DECL FDAT FP437={TOOL_NO 1,BASE_NO 1,IPO_FRAME #BASE,POINT2[] " ",TQ_STATE FALSE}
DECL E6POS XP437={X 1259.09706,Y 164.02997,Z 815.2861,A 180,B 0,C -180,S 2,T 2,E1 0,E2 0,E3 0,E4 0,E5 0,E6 0}
DECL PDAT PPDATP96={VEL 100,ACC 100,APO_DIST 100,APO_MODE #CDIS,GEAR_JERK 100.000,EXAX_IGN 0}
DECL FDAT FP33={TOOL_NO 1,BASE_NO 1,IPO_FRAME #BASE,POINT2[] " ",TQ_STATE FALSE}
DECL E6POS XP33={X 427.07288,Y -471.93323,Z 1236.2934,A 180,B 0,C 180,S 2,T 2,E1 0,E2 0,E3 0,E4 0,E5 0,E6 0}
DECL LDAT LCPDATP186={VEL 1,ACC 100,APO_DIST 100,APO_FAC 50.0,ORI_TYP #VAR,CIRC_TYP #BASE,JERK_FAC 50.0}
DECL FDAT FP31={TOOL_NO 1,BASE_NO 1,IPO_FRAME #BASE,POINT2[] " ",TQ_STATE FALSE}
DECL E6POS XP31={X 427.07317,Y -471.93292,Z 1136.29359,A -180,B 0,C 180,S 2,T 2,E1 0,E2 0,E3 0,E4 0,E5 0,E6 0}
DECL LDAT LCPDATP187={VEL 1,ACC 100,APO_DIST 100,APO_FAC 50.0,ORI_TYP #VAR,CIRC_TYP #BASE,JERK_FAC 50.0}
DECL FDAT FP32={TOOL_NO 1,BASE_NO 1,IPO_FRAME #BASE,POINT2[] " ",TQ_STATE FALSE}
DECL E6POS XP32={X 377.07317,Y -471.93292,Z 1036.29359,A -180,B 0,C 180,S 2,T 2,E1 0,E2 0,E3 0,E4 0,E5 0,E6 0}
; DECL PDAT PPDATP96={VEL 100,ACC 100,APO_DIST 100,APO_MODE #CDIS,GEAR_JERK 100.000,EXAX_IGN 0}
DECL FDAT FP273={TOOL_NO 1,BASE_NO 1,IPO_FRAME #BASE,POINT2[] " ",TQ_STATE FALSE}
DECL E6POS XP273={X 745.07288,Y -471.93323,Z 1236.2934,A 180,B 0,C 180,S 2,T 2,E1 0,E2 0,E3 0,E4 0,E5 0,E6 0}
; DECL LDAT LCPDATP186={VEL 1,ACC 100,APO_DIST 100,APO_FAC 50.0,ORI_TYP #VAR,CIRC_TYP #BASE,JERK_FAC 50.0}
DECL FDAT FP274={TOOL_NO 1,BASE_NO 1,IPO_FRAME #BASE,POINT2[] " ",TQ_STATE FALSE}
DECL E6POS XP274={X 745.07317,Y -471.93292,Z 1136.29359,A -180,B 0,C 180,S 2,T 2,E1 0,E2 0,E3 0,E4 0,E5 0,E6 0}
; DECL LDAT LCPDATP187={VEL 1,ACC 100,APO_DIST 100,APO_FAC 50.0,ORI_TYP #VAR,CIRC_TYP #BASE,JERK_FAC 50.0}
DECL FDAT FP275={TOOL_NO 1,BASE_NO 1,IPO_FRAME #BASE,POINT2[] " ",TQ_STATE FALSE}
DECL E6POS XP275={X 695.07317,Y -471.93292,Z 1036.29359,A -180,B 0,C 180,S 2,T 2,E1 0,E2 0,E3 0,E4 0,E5 0,E6 0}
DECL PDAT PPDATP97={VEL 100,ACC 100,APO_DIST 100,APO_MODE #CDIS,GEAR_JERK 100.000,EXAX_IGN 0}
DECL FDAT FP278={TOOL_NO 1,BASE_NO 1,IPO_FRAME #BASE,POINT2[] " ",TQ_STATE FALSE}
DECL E6POS XP278={X 537.09939,Y -651.74884,Z 1306.29683,A 90,B 0,C 180,S 2,T 2,E1 0,E2 0,E3 0,E4 0,E5 0,E6 0}
DECL LDAT LCPDATP188={VEL 1,ACC 100,APO_DIST 100,APO_FAC 50.0,ORI_TYP #VAR,CIRC_TYP #BASE,JERK_FAC 50.0}
DECL FDAT FP276={TOOL_NO 1,BASE_NO 1,IPO_FRAME #BASE,POINT2[] " ",TQ_STATE FALSE}
DECL E6POS XP276={X 537.09936,Y -651.74901,Z 1136.29687,A 90,B 0,C 180,S 2,T 2,E1 0,E2 0,E3 0,E4 0,E5 0,E6 0}
DECL LDAT LCPDATP189={VEL 1,ACC 100,APO_DIST 100,APO_FAC 50.0,ORI_TYP #VAR,CIRC_TYP #BASE,JERK_FAC 50.0}
DECL FDAT FP277={TOOL_NO 1,BASE_NO 1,IPO_FRAME #BASE,POINT2[] " ",TQ_STATE FALSE}
DECL E6POS XP277={X 537.0999,Y -701.74921,Z 1036.29638,A 90,B 0,C -180,S 2,T 2,E1 0,E2 0,E3 0,E4 0,E5 0,E6 0}
; DECL PDAT PPDATP97={VEL 100,ACC 100,APO_DIST 100,APO_MODE #CDIS,GEAR_JERK 100.000,EXAX_IGN 0}
DECL FDAT FP279={TOOL_NO 1,BASE_NO 1,IPO_FRAME #BASE,POINT2[] " ",TQ_STATE FALSE}
DECL E6POS XP279={X 537.09939,Y -333.74884,Z 1306.29683,A 90,B 0,C 180,S 2,T 2,E1 0,E2 0,E3 0,E4 0,E5 0,E6 0}
; DECL LDAT LCPDATP188={VEL 1,ACC 100,APO_DIST 100,APO_FAC 50.0,ORI_TYP #VAR,CIRC_TYP #BASE,JERK_FAC 50.0}
DECL FDAT FP280={TOOL_NO 1,BASE_NO 1,IPO_FRAME #BASE,POINT2[] " ",TQ_STATE FALSE}
DECL E6POS XP280={X 537.09936,Y -333.74901,Z 1136.29687,A 90,B 0,C 180,S 2,T 2,E1 0,E2 0,E3 0,E4 0,E5 0,E6 0}
; DECL LDAT LCPDATP189={VEL 1,ACC 100,APO_DIST 100,APO_FAC 50.0,ORI_TYP #VAR,CIRC_TYP #BASE,JERK_FAC 50.0}
DECL FDAT FP281={TOOL_NO 1,BASE_NO 1,IPO_FRAME #BASE,POINT2[] " ",TQ_STATE FALSE}
DECL E6POS XP281={X 537.0999,Y -383.74921,Z 1036.29638,A 90,B 0,C -180,S 2,T 2,E1 0,E2 0,E3 0,E4 0,E5 0,E6 0}
; DECL PDAT PPDATP97={VEL 100,ACC 100,APO_DIST 100,APO_MODE #CDIS,GEAR_JERK 100.000,EXAX_IGN 0}
DECL FDAT FP282={TOOL_NO 1,BASE_NO 1,IPO_FRAME #BASE,POINT2[] " ",TQ_STATE FALSE}
DECL E6POS XP282={X 1223.09936,Y -1027.74903,Z 1306.29661,A 90,B 0,C 180,S 2,T 34,E1 0,E2 0,E3 0,E4 0,E5 0,E6 0}
; DECL LDAT LCPDATP188={VEL 1,ACC 100,APO_DIST 100,APO_FAC 50.0,ORI_TYP #VAR,CIRC_TYP #BASE,JERK_FAC 50.0}
DECL FDAT FP283={TOOL_NO 1,BASE_NO 1,IPO_FRAME #BASE,POINT2[] " ",TQ_STATE FALSE}
DECL E6POS XP283={X 1223.09936,Y -1027.74901,Z 1136.29687,A 90,B 0,C 180,S 2,T 34,E1 0,E2 0,E3 0,E4 0,E5 0,E6 0}
; DECL LDAT LCPDATP189={VEL 1,ACC 100,APO_DIST 100,APO_FAC 50.0,ORI_TYP #VAR,CIRC_TYP #BASE,JERK_FAC 50.0}
DECL FDAT FP284={TOOL_NO 1,BASE_NO 1,IPO_FRAME #BASE,POINT2[] " ",TQ_STATE FALSE}
DECL E6POS XP284={X 1173.0999,Y -1077.74921,Z 1036.29638,A 90,B 0,C -180,S 2,T 34,E1 0,E2 0,E3 0,E4 0,E5 0,E6 0}
; DECL PDAT PPDATP97={VEL 100,ACC 100,APO_DIST 100,APO_MODE #CDIS,GEAR_JERK 100.000,EXAX_IGN 0}
DECL FDAT FP285={TOOL_NO 1,BASE_NO 1,IPO_FRAME #BASE,POINT2[] " ",TQ_STATE FALSE}
DECL E6POS XP285={X 1223.09936,Y -709.74905,Z 1306.29686,A 90,B 0,C 180,S 2,T 34,E1 0,E2 0,E3 0,E4 0,E5 0,E6 0}
; DECL LDAT LCPDATP188={VEL 1,ACC 100,APO_DIST 100,APO_FAC 50.0,ORI_TYP #VAR,CIRC_TYP #BASE,JERK_FAC 50.0}
DECL FDAT FP286={TOOL_NO 1,BASE_NO 1,IPO_FRAME #BASE,POINT2[] " ",TQ_STATE FALSE}
DECL E6POS XP286={X 1223.09936,Y -709.74901,Z 1136.29687,A 90,B 0,C 180,S 2,T 34,E1 0,E2 0,E3 0,E4 0,E5 0,E6 0}
; DECL LDAT LCPDATP189={VEL 1,ACC 100,APO_DIST 100,APO_FAC 50.0,ORI_TYP #VAR,CIRC_TYP #BASE,JERK_FAC 50.0}
DECL FDAT FP287={TOOL_NO 1,BASE_NO 1,IPO_FRAME #BASE,POINT2[] " ",TQ_STATE FALSE}
DECL E6POS XP287={X 1173.0999,Y -759.74921,Z 1036.29638,A 90,B 0,C -180,S 2,T 34,E1 0,E2 0,E3 0,E4 0,E5 0,E6 0}
; DECL PDAT PPDATP86={VEL 100,ACC 100,APO_DIST 100,APO_MODE #CDIS,GEAR_JERK 100.000,EXAX_IGN 0}
DECL FDAT FP438={TOOL_NO 1,BASE_NO 1,IPO_FRAME #BASE,POINT2[] " ",TQ_STATE FALSE}
DECL E6POS XP438={X 981.09733,Y 214.03031,Z 1286.28573,A 180,B 0,C 180,S 2,T 2,E1 0,E2 0,E3 0,E4 0,E5 0,E6 0}
; DECL LDAT LCPDATP173={VEL 1,ACC 100,APO_DIST 100,APO_FAC 50.0,ORI_TYP #VAR,CIRC_TYP #BASE,JERK_FAC 50.0}
DECL FDAT FP439={TOOL_NO 1,BASE_NO 1,IPO_FRAME #BASE,POINT2[] " ",TQ_STATE FALSE}
DECL E6POS XP439={X 981.09706,Y 214.03031,Z 1186.28614,A 180,B 0,C -180,S 2,T 2,E1 0,E2 0,E3 0,E4 0,E5 0,E6 0}
; DECL LDAT LCPDATP172={VEL 1,ACC 100,APO_DIST 100,APO_FAC 50.0,ORI_TYP #VAR,CIRC_TYP #BASE,JERK_FAC 50.0}
DECL FDAT FP440={TOOL_NO 1,BASE_NO 1,IPO_FRAME #BASE,POINT2[] " ",TQ_STATE FALSE}
DECL E6POS XP440={X 941.09706,Y 164.02997,Z 1036.2861,A 180,B 0,C -180,S 2,T 2,E1 0,E2 0,E3 0,E4 0,E5 0,E6 0}
; DECL PDAT PPDATP86={VEL 100,ACC 100,APO_DIST 100,APO_MODE #CDIS,GEAR_JERK 100.000,EXAX_IGN 0}
DECL FDAT FP453={TOOL_NO 1,BASE_NO 1,IPO_FRAME #BASE,POINT2[] " ",TQ_STATE FALSE}
DECL E6POS XP453={X 1299.09733,Y 214.03031,Z 1286.28573,A 180,B 0,C 180,S 2,T 2,E1 0,E2 0,E3 0,E4 0,E5 0,E6 0}
; DECL LDAT LCPDATP173={VEL 1,ACC 100,APO_DIST 100,APO_FAC 50.0,ORI_TYP #VAR,CIRC_TYP #BASE,JERK_FAC 50.0}
DECL FDAT FP454={TOOL_NO 1,BASE_NO 1,IPO_FRAME #BASE,POINT2[] " ",TQ_STATE FALSE}
DECL E6POS XP454={X 1299.09706,Y 214.03031,Z 1186.28614,A 180,B 0,C -180,S 2,T 2,E1 0,E2 0,E3 0,E4 0,E5 0,E6 0}
; DECL LDAT LCPDATP172={VEL 1,ACC 100,APO_DIST 100,APO_FAC 50.0,ORI_TYP #VAR,CIRC_TYP #BASE,JERK_FAC 50.0}
DECL FDAT FP455={TOOL_NO 1,BASE_NO 1,IPO_FRAME #BASE,POINT2[] " ",TQ_STATE FALSE}
DECL E6POS XP455={X 1259.09706,Y 164.02997,Z 1036.2861,A 180,B 0,C -180,S 2,T 2,E1 0,E2 0,E3 0,E4 0,E5 0,E6 0}
; ENDDAT for Mtrz_P1_7Aero
; Data for DepositoAll
; ENDDAT for DepositoAll
; Data for Mtrz_P1_32BarPacking
DECL PDAT PPDATP22={VEL 100,ACC 100,APO_DIST 100,APO_MODE #CDIS,GEAR_JERK 100.000,EXAX_IGN 0}
DECL FDAT FP93={TOOL_NO 1,BASE_NO 1,IPO_FRAME #BASE,POINT2[] " ",TQ_STATE FALSE}
DECL E6POS XP93={X 1072.98685,Y -436.50081,Z 1272.32323,A 180,B 0,C -180,S 2,T 2,E1 0,E2 0,E3 0,E4 0,E5 0,E6 0}
DECL LDAT LCPDATP42={VEL 1,ACC 100,APO_DIST 100,APO_FAC 50.0,ORI_TYP #VAR,CIRC_TYP #BASE,JERK_FAC 50.0}
DECL FDAT FP94={TOOL_NO 1,BASE_NO 1,IPO_FRAME #BASE,POINT2[] " ",TQ_STATE FALSE}
DECL E6POS XP94={X 1072.98689,Y -436.50116,Z 1122.32295,A 180,B 0,C -180,S 2,T 2,E1 0,E2 0,E3 0,E4 0,E5 0,E6 0}
DECL LDAT LCPDATP43={VEL 1,ACC 100,APO_DIST 100,APO_FAC 50.0,ORI_TYP #VAR,CIRC_TYP #BASE,JERK_FAC 50.0}
DECL FDAT FP95={TOOL_NO 1,BASE_NO 1,IPO_FRAME #BASE,POINT2[] " ",TQ_STATE FALSE}
DECL E6POS XP95={X 1172.98673,Y -436.50078,Z 872.32277,A 180,B 0,C -180,S 2,T 2,E1 0,E2 0,E3 0,E4 0,E5 0,E6 0}
DECL PDAT PPDATP23={VEL 100,ACC 100,APO_DIST 100,APO_MODE #CDIS,GEAR_JERK 100.000,EXAX_IGN 0}
DECL FDAT FP96={TOOL_NO 1,BASE_NO 1,IPO_FRAME #BASE,POINT2[] " ",TQ_STATE FALSE}
DECL E6POS XP96={X 681.98616,Y -436.50075,Z 1272.32295,A 180,B 0,C 180,S 2,T 2,E1 0,E2 0,E3 0,E4 0,E5 0,E6 0}
DECL LDAT LCPDATP45={VEL 1,ACC 100,APO_DIST 100,APO_FAC 50.0,ORI_TYP #VAR,CIRC_TYP #BASE,JERK_FAC 50.0}
DECL FDAT FP98={TOOL_NO 1,BASE_NO 1,IPO_FRAME #BASE,POINT2[] " ",TQ_STATE FALSE}
DECL E6POS XP98={X 681.98616,Y -436.50081,Z 1122.3233,A -180,B 0,C -180,S 2,T 2,E1 0,E2 0,E3 0,E4 0,E5 0,E6 0}
DECL LDAT LCPDATP44={VEL 1,ACC 100,APO_DIST 100,APO_FAC 50.0,ORI_TYP #VAR,CIRC_TYP #BASE,JERK_FAC 50.0}
DECL FDAT FP97={TOOL_NO 1,BASE_NO 1,IPO_FRAME #BASE,POINT2[] " ",TQ_STATE FALSE}
DECL E6POS XP97={X 781.9869,Y -436.50077,Z 872.32219,A 180,B 0,C 180,S 2,T 2,E1 0,E2 0,E3 0,E4 0,E5 0,E6 0}
DECL PDAT PPDATP24={VEL 100,ACC 100,APO_DIST 100,APO_MODE #CDIS,GEAR_JERK 100.000,EXAX_IGN 0}
DECL FDAT FP99={TOOL_NO 1,BASE_NO 1,IPO_FRAME #BASE,POINT2[] " ",TQ_STATE FALSE}
DECL E6POS XP99={X 290.98674,Y -436.50102,Z 1272.32359,A -180,B 0,C -180,S 2,T 2,E1 0,E2 0,E3 0,E4 0,E5 0,E6 0}
DECL LDAT LCPDATP46={VEL 1,ACC 100,APO_DIST 100,APO_FAC 50.0,ORI_TYP #VAR,CIRC_TYP #BASE,JERK_FAC 50.0}
DECL FDAT FP100={TOOL_NO 1,BASE_NO 1,IPO_FRAME #BASE,POINT2[] " ",TQ_STATE FALSE}
DECL E6POS XP100={X 290.9867,Y -436.50113,Z 1122.32278,A 180,B 0,C 180,S 2,T 2,E1 0,E2 0,E3 0,E4 0,E5 0,E6 0}
DECL LDAT LCPDATP47={VEL 1,ACC 100,APO_DIST 100,APO_FAC 50.0,ORI_TYP #VAR,CIRC_TYP #BASE,JERK_FAC 50.0}
DECL FDAT FP101={TOOL_NO 1,BASE_NO 1,IPO_FRAME #BASE,POINT2[] " ",TQ_STATE FALSE}
DECL E6POS XP101={X 390.98701,Y -436.50118,Z 872.32277,A 180,B 0,C 180,S 2,T 2,E1 0,E2 0,E3 0,E4 0,E5 0,E6 0}
; ENDDAT for Mtrz_P1_32BarPacking
; Data for Mtrz_P1_33BarPacking
DECL PDAT PPDATP25={VEL 100,ACC 100,APO_DIST 100,APO_MODE #CDIS,GEAR_JERK 100.000,EXAX_IGN 0}
DECL FDAT FP102={TOOL_NO 1,BASE_NO 1,IPO_FRAME #BASE,POINT2[] " ",TQ_STATE FALSE}
DECL E6POS XP102={X 1047.81428,Y -467.93231,Z 1263.51475,A 180,B 0,C 180,S 2,T 2,E1 0,E2 0,E3 0,E4 0,E5 0,E6 0}
DECL LDAT LCPDATP48={VEL 1,ACC 100,APO_DIST 100,APO_FAC 50.0,ORI_TYP #VAR,CIRC_TYP #BASE,JERK_FAC 50.0}
DECL FDAT FP103={TOOL_NO 1,BASE_NO 1,IPO_FRAME #BASE,POINT2[] " ",TQ_STATE FALSE}
DECL E6POS XP103={X 1047.81429,Y -467.93247,Z 1063.51485,A 180,B 0,C 180,S 2,T 2,E1 0,E2 0,E3 0,E4 0,E5 0,E6 0}
DECL LDAT LCPDATP49={VEL 1,ACC 100,APO_DIST 100,APO_FAC 50.0,ORI_TYP #VAR,CIRC_TYP #BASE,JERK_FAC 50.0}
DECL FDAT FP104={TOOL_NO 1,BASE_NO 1,IPO_FRAME #BASE,POINT2[] " ",TQ_STATE FALSE}
DECL E6POS XP104={X 1147.81449,Y -467.93244,Z 863.51516,A 180,B 0,C 180,S 2,T 2,E1 0,E2 0,E3 0,E4 0,E5 0,E6 0}
DECL PDAT PPDATP26={VEL 100,ACC 100,APO_DIST 100,APO_MODE #CDIS,GEAR_JERK 100.000,EXAX_IGN 0}
DECL FDAT FP105={TOOL_NO 1,BASE_NO 1,IPO_FRAME #BASE,POINT2[] " ",TQ_STATE FALSE}
DECL E6POS XP105={X 482.81507,Y -467.93234,Z 1263.51544,A 180,B 0,C 180,S 2,T 2,E1 0,E2 0,E3 0,E4 0,E5 0,E6 0}
DECL LDAT LCPDATP50={VEL 1,ACC 100,APO_DIST 100,APO_FAC 50.0,ORI_TYP #VAR,CIRC_TYP #BASE,JERK_FAC 50.0}
DECL FDAT FP106={TOOL_NO 1,BASE_NO 1,IPO_FRAME #BASE,POINT2[] " ",TQ_STATE FALSE}
DECL E6POS XP106={X 482.81509,Y -467.93223,Z 1063.51535,A 180,B 0,C 180,S 2,T 2,E1 0,E2 0,E3 0,E4 0,E5 0,E6 0}
DECL LDAT LCPDATP51={VEL 1,ACC 100,APO_DIST 100,APO_FAC 50.0,ORI_TYP #VAR,CIRC_TYP #BASE,JERK_FAC 50.0}
DECL FDAT FP107={TOOL_NO 1,BASE_NO 1,IPO_FRAME #BASE,POINT2[] " ",TQ_STATE FALSE}
DECL E6POS XP107={X 582.81489,Y -467.93218,Z 863.51495,A -180,B 0,C 180,S 2,T 2,E1 0,E2 0,E3 0,E4 0,E5 0,E6 0}
; ENDDAT for Mtrz_P1_33BarPacking
; Data for Mtrz_P1_37BarPacking
DECL PDAT PPDATP19={VEL 100,ACC 100,APO_DIST 100,APO_MODE #CDIS,GEAR_JERK 100.000,EXAX_IGN 0}
DECL FDAT FP80={TOOL_NO 1,BASE_NO 1,IPO_FRAME #BASE,POINT2[] " ",TQ_STATE FALSE}
DECL E6POS XP80={X 553.8887,Y -887.44398,Z 1263.48448,A 90,B 0,C 180,S 2,T 2,E1 0,E2 0,E3 0,E4 0,E5 0,E6 0}
DECL LDAT LCPDATP36={VEL 1,ACC 100,APO_DIST 100,APO_FAC 50.0,ORI_TYP #VAR,CIRC_TYP #BASE,JERK_FAC 50.0}
DECL FDAT FP81={TOOL_NO 1,BASE_NO 1,IPO_FRAME #BASE,POINT2[] " ",TQ_STATE FALSE}
DECL E6POS XP81={X 553.88871,Y -887.44391,Z 1063.48533,A 90,B 0,C 180,S 2,T 2,E1 0,E2 0,E3 0,E4 0,E5 0,E6 0}
DECL LDAT LCPDATP37={VEL 1,ACC 100,APO_DIST 100,APO_FAC 50.0,ORI_TYP #VAR,CIRC_TYP #BASE,JERK_FAC 50.0}
DECL FDAT FP82={TOOL_NO 1,BASE_NO 1,IPO_FRAME #BASE,POINT2[] " ",TQ_STATE FALSE}
DECL E6POS XP82={X 553.88862,Y -987.4438,Z 863.48478,A 90,B 0,C 180,S 2,T 2,E1 0,E2 0,E3 0,E4 0,E5 0,E6 0}
DECL PDAT PPDATP20={VEL 100,ACC 100,APO_DIST 100,APO_MODE #CDIS,GEAR_JERK 100.000,EXAX_IGN 0}
DECL FDAT FP83={TOOL_NO 1,BASE_NO 1,IPO_FRAME #BASE,POINT2[] " ",TQ_STATE FALSE}
DECL E6POS XP83={X 553.88861,Y -391.44429,Z 1263.48465,A 90,B 0,C 180,S 2,T 2,E1 0,E2 0,E3 0,E4 0,E5 0,E6 0}
DECL LDAT LCPDATP38={VEL 1,ACC 100,APO_DIST 100,APO_FAC 50.0,ORI_TYP #VAR,CIRC_TYP #BASE,JERK_FAC 50.0}
DECL FDAT FP84={TOOL_NO 1,BASE_NO 1,IPO_FRAME #BASE,POINT2[] " ",TQ_STATE FALSE}
DECL E6POS XP84={X 553.88866,Y -391.44397,Z 1063.48492,A 90,B 0,C -180,S 2,T 2,E1 0,E2 0,E3 0,E4 0,E5 0,E6 0}
DECL LDAT LCPDATP39={VEL 1,ACC 100,APO_DIST 100,APO_FAC 50.0,ORI_TYP #VAR,CIRC_TYP #BASE,JERK_FAC 50.0}
DECL FDAT FP85={TOOL_NO 1,BASE_NO 1,IPO_FRAME #BASE,POINT2[] " ",TQ_STATE FALSE}
DECL E6POS XP85={X 553.88842,Y -491.44382,Z 863.48495,A 90,B 0,C 180,S 2,T 2,E1 0,E2 0,E3 0,E4 0,E5 0,E6 0}
; ENDDAT for Mtrz_P1_37BarPacking
; Data for Mtrz_P1_36BarPacking
DECL PDAT PPDATP21={VEL 100,ACC 100,APO_DIST 100,APO_MODE #CDIS,GEAR_JERK 100.000,EXAX_IGN 0}
DECL FDAT FP86={TOOL_NO 1,BASE_NO 1,IPO_FRAME #BASE,POINT2[] " ",TQ_STATE FALSE}
DECL E6POS XP86={X 558.59091,Y -644.52527,Z 1263.46025,A 90,B 0,C 180,S 2,T 2,E1 0,E2 0,E3 0,E4 0,E5 0,E6 0}
DECL LDAT LCPDATP40={VEL 1,ACC 100,APO_DIST 100,APO_FAC 50.0,ORI_TYP #VAR,CIRC_TYP #BASE,JERK_FAC 50.0}
DECL FDAT FP87={TOOL_NO 1,BASE_NO 1,IPO_FRAME #BASE,POINT2[] " ",TQ_STATE FALSE}
DECL E6POS XP87={X 558.59085,Y -644.52561,Z 1063.45997,A 90,B 0,C -180,S 2,T 2,E1 0,E2 0,E3 0,E4 0,E5 0,E6 0}
DECL LDAT LCPDATP41={VEL 1,ACC 100,APO_DIST 100,APO_FAC 50.0,ORI_TYP #VAR,CIRC_TYP #BASE,JERK_FAC 50.0}
DECL FDAT FP88={TOOL_NO 1,BASE_NO 1,IPO_FRAME #BASE,POINT2[] " ",TQ_STATE FALSE}
DECL E6POS XP88={X 558.59062,Y -744.5248,Z 863.45988,A 90,B 0,C 180,S 2,T 2,E1 0,E2 0,E3 0,E4 0,E5 0,E6 0}
; ENDDAT for Mtrz_P1_36BarPacking
; Data for Mtrz_P1_34BarPacking
DECL PDAT PPDATP27={VEL 100,ACC 100,APO_DIST 100,APO_MODE #CDIS,GEAR_JERK 100.000,EXAX_IGN 0}
DECL FDAT FP108={TOOL_NO 1,BASE_NO 1,IPO_FRAME #BASE,POINT2[] " ",TQ_STATE FALSE}
DECL E6POS XP108={X 1055.40907,Y -256.77745,Z 1034.57222,A 180,B 0,C -180,S 2,T 2,E1 0,E2 0,E3 0,E4 0,E5 0,E6 0}
DECL LDAT LCPDATP52={VEL 1,ACC 100,APO_DIST 100,APO_FAC 50.0,ORI_TYP #VAR,CIRC_TYP #BASE,JERK_FAC 50.0}
DECL FDAT FP109={TOOL_NO 1,BASE_NO 1,IPO_FRAME #BASE,POINT2[] " ",TQ_STATE FALSE}
DECL E6POS XP109={X 1055.40912,Y -256.77793,Z 914.57188,A -180,B 0,C -180,S 2,T 2,E1 0,E2 0,E3 0,E4 0,E5 0,E6 0}
DECL LDAT LCPDATP53={VEL 1,ACC 100,APO_DIST 100,APO_FAC 50.0,ORI_TYP #VAR,CIRC_TYP #BASE,JERK_FAC 50.0}
DECL FDAT FP110={TOOL_NO 1,BASE_NO 1,IPO_FRAME #BASE,POINT2[] " ",TQ_STATE FALSE}
DECL E6POS XP110={X 1155.40894,Y -256.77773,Z 814.57153,A -180,B 0,C 180,S 2,T 2,E1 0,E2 0,E3 0,E4 0,E5 0,E6 0}
DECL PDAT PPDATP29={VEL 100,ACC 100,APO_DIST 100,APO_MODE #CDIS,GEAR_JERK 100.000,EXAX_IGN 0}
DECL FDAT FP118={TOOL_NO 1,BASE_NO 1,IPO_FRAME #BASE,POINT2[] " ",TQ_STATE FALSE}
DECL E6POS XP118={X 516.40827,Y -256.77794,Z 1034.57222,A -180,B 0,C -180,S 2,T 2,E1 0,E2 0,E3 0,E4 0,E5 0,E6 0}
DECL LDAT LCPDATP54={VEL 1,ACC 100,APO_DIST 100,APO_FAC 50.0,ORI_TYP #VAR,CIRC_TYP #BASE,JERK_FAC 50.0}
DECL FDAT FP116={TOOL_NO 1,BASE_NO 1,IPO_FRAME #BASE,POINT2[] " ",TQ_STATE FALSE}
DECL E6POS XP116={X 516.40827,Y -256.77795,Z 914.57211,A -180,B 0,C -180,S 2,T 2,E1 0,E2 0,E3 0,E4 0,E5 0,E6 0}
DECL LDAT LCPDATP55={VEL 1,ACC 100,APO_DIST 100,APO_FAC 50.0,ORI_TYP #VAR,CIRC_TYP #BASE,JERK_FAC 50.0}
DECL FDAT FP117={TOOL_NO 1,BASE_NO 1,IPO_FRAME #BASE,POINT2[] " ",TQ_STATE FALSE}
DECL E6POS XP117={X 586.40852,Y -256.7776,Z 814.57168,A 180,B 0,C 180,S 2,T 2,E1 0,E2 0,E3 0,E4 0,E5 0,E6 0}
; ENDDAT for Mtrz_P1_34BarPacking
; Data for Mtrz_P1_35BarPacking
DECL PDAT PPDATP47={VEL 100,ACC 100,APO_DIST 100,APO_MODE #CDIS,GEAR_JERK 100.000,EXAX_IGN 0}
DECL FDAT FP188={TOOL_NO 1,BASE_NO 1,IPO_FRAME #BASE,POINT2[] " ",TQ_STATE FALSE}
DECL E6POS XP188={X 1128.19617,Y -447.20835,Z 1215.66349,A 180,B 0,C 180,S 2,T 2,E1 0,E2 0,E3 0,E4 0,E5 0,E6 0}
DECL LDAT LCPDATP92={VEL 1,ACC 100,APO_DIST 100,APO_FAC 50.0,ORI_TYP #VAR,CIRC_TYP #BASE,JERK_FAC 50.0}
DECL FDAT FP189={TOOL_NO 1,BASE_NO 1,IPO_FRAME #BASE,POINT2[] " ",TQ_STATE FALSE}
DECL E6POS XP189={X 1128.19623,Y -447.20835,Z 1015.66288,A 180,B 0,C 180,S 2,T 2,E1 0,E2 0,E3 0,E4 0,E5 0,E6 0}
DECL LDAT LCPDATP93={VEL 1,ACC 100,APO_DIST 100,APO_FAC 50.0,ORI_TYP #VAR,CIRC_TYP #BASE,JERK_FAC 50.0}
DECL FDAT FP190={TOOL_NO 1,BASE_NO 1,IPO_FRAME #BASE,POINT2[] " ",TQ_STATE FALSE}
DECL E6POS XP190={X 1178.19625,Y -447.20835,Z 865.66289,A -180,B 0,C -180,S 2,T 2,E1 0,E2 0,E3 0,E4 0,E5 0,E6 0}
DECL PDAT PPDATP48={VEL 100,ACC 100,APO_DIST 100,APO_MODE #CDIS,GEAR_JERK 100.000,EXAX_IGN 0}
DECL FDAT FP193={TOOL_NO 1,BASE_NO 1,IPO_FRAME #BASE,POINT2[] " ",TQ_STATE FALSE}
DECL E6POS XP193={X 532.19563,Y -447.20805,Z 1215.66362,A -180,B 0,C -180,S 2,T 2,E1 0,E2 0,E3 0,E4 0,E5 0,E6 0}
DECL LDAT LCPDATP95={VEL 1,ACC 100,APO_DIST 100,APO_FAC 50.0,ORI_TYP #VAR,CIRC_TYP #BASE,JERK_FAC 50.0}
DECL FDAT FP192={TOOL_NO 1,BASE_NO 1,IPO_FRAME #BASE,POINT2[] " ",TQ_STATE FALSE}
DECL E6POS XP192={X 532.19539,Y -447.20804,Z 1015.66268,A -180,B 0,C -180,S 2,T 2,E1 0,E2 0,E3 0,E4 0,E5 0,E6 0}
DECL LDAT LCPDATP94={VEL 1,ACC 100,APO_DIST 100,APO_FAC 50.0,ORI_TYP #VAR,CIRC_TYP #BASE,JERK_FAC 50.0}
DECL FDAT FP191={TOOL_NO 1,BASE_NO 1,IPO_FRAME #BASE,POINT2[] " ",TQ_STATE FALSE}
DECL E6POS XP191={X 582.19539,Y -447.20804,Z 865.66281,A -180,B 0,C 180,S 2,T 2,E1 0,E2 0,E3 0,E4 0,E5 0,E6 0}
DECL PDAT PPDATP49={VEL 100,ACC 100,APO_DIST 100,APO_MODE #CDIS,GEAR_JERK 100.000,EXAX_IGN 0}
DECL FDAT FP194={TOOL_NO 1,BASE_NO 1,IPO_FRAME #BASE,POINT2[] " ",TQ_STATE FALSE}
DECL E6POS XP194={X 561.78309,Y -442.05433,Z 1274.46292,A 90,B 0,C 180,S 2,T 2,E1 0,E2 0,E3 0,E4 0,E5 0,E6 0}
DECL LDAT LCPDATP96={VEL 1,ACC 100,APO_DIST 100,APO_FAC 50.0,ORI_TYP #VAR,CIRC_TYP #BASE,JERK_FAC 50.0}
DECL FDAT FP195={TOOL_NO 1,BASE_NO 1,IPO_FRAME #BASE,POINT2[] " ",TQ_STATE FALSE}
DECL E6POS XP195={X 561.78309,Y -442.05406,Z 1024.46338,A 90,B 0,C 180,S 2,T 2,E1 0,E2 0,E3 0,E4 0,E5 0,E6 0}
DECL LDAT LCPDATP97={VEL 1,ACC 100,APO_DIST 100,APO_FAC 50.0,ORI_TYP #VAR,CIRC_TYP #BASE,JERK_FAC 50.0}
DECL FDAT FP196={TOOL_NO 1,BASE_NO 1,IPO_FRAME #BASE,POINT2[] " ",TQ_STATE FALSE}
DECL E6POS XP196={X 561.78309,Y -589.19041,Z 865.6383,A 90,B 0,C -180,S 2,T 2,E1 0,E2 0,E3 0,E4 0,E5 0,E6 0}
; ENDDAT for Mtrz_P1_35BarPacking
; Data for ConfGarraOp0
; ENDDAT for ConfGarraOp0
; Data for FechaGarraOp0
; ENDDAT for FechaGarraOp0
; Data for AbreGarraOp0
; ENDDAT for AbreGarraOp0
; Data for PickCaixasSimulador
; ENDDAT for PickCaixasSimulador
; Data for ConfGarraOp1
; ENDDAT for ConfGarraOp1
; Data for Pick_E_1_P_2
; DECL PDAT PPDATP1={VEL 100,ACC 100,APO_DIST 100,APO_MODE #CDIS,GEAR_JERK 100.000,EXAX_IGN 0}
DECL FDAT FP76={TOOL_NO 1,BASE_NO 3,IPO_FRAME #BASE,POINT2[] " ",TQ_STATE FALSE}
DECL E6POS XP76={X 548.60753,Y -2.83256,Z 2105.79953,A 90,B 0,C -180,S 2,T 34,E1 0,E2 0,E3 0,E4 0,E5 0,E6 0}
; DECL LDAT LCPDATP2={VEL 1,ACC 100,APO_DIST 100,APO_FAC 50.0,ORI_TYP #VAR,CIRC_TYP #BASE,JERK_FAC 50.0}
DECL FDAT FP77={TOOL_NO 1,BASE_NO 3,IPO_FRAME #BASE,POINT2[] " ",TQ_STATE FALSE}
DECL E6POS XP77={X 548.60753,Y -2.8321,Z 1392.47867,A 90,B 0,C -180,S 2,T 34,E1 0,E2 0,E3 0,E4 0,E5 0,E6 0}
; DECL LDAT LCPDATP1={VEL 1,ACC 100,APO_DIST 100,APO_FAC 50.0,ORI_TYP #VAR,CIRC_TYP #BASE,JERK_FAC 50.0}
DECL FDAT FPick_E_1_P_2={TOOL_NO 1,BASE_NO 3,IPO_FRAME #BASE,POINT2[] " ",TQ_STATE FALSE}
DECL E6POS XPick_E_1_P_2={X 548.60753,Y 19.40185,Z 1392.47867,A 90,B 0,C -180,S 2,T 34,E1 0,E2 0,E3 0,E4 0,E5 0,E6 0}
; DECL LDAT LCPDATP3={VEL 1,ACC 100,APO_DIST 100,APO_FAC 50.0,ORI_TYP #VAR,CIRC_TYP #BASE,JERK_FAC 50.0}
DECL FDAT FP79={TOOL_NO 1,BASE_NO 3,IPO_FRAME #BASE,POINT2[] " ",TQ_STATE FALSE}
DECL E6POS XP79={X 548.60753,Y 19.40185,Z 2105.80057,A 90,B 0,C 180,S 2,T 34,E1 0,E2 0,E3 0,E4 0,E5 0,E6 0}
; ENDDAT for Pick_E_1_P_2
; Data for ConfGarraOp2
; ENDDAT for ConfGarraOp2
; Data for ConfGarraOp3
; ENDDAT for ConfGarraOp3
; Data for Pick_E_1_P_3
; DECL PDAT PPDATP1={VEL 100,ACC 100,APO_DIST 100,APO_MODE #CDIS,GEAR_JERK 100.000,EXAX_IGN 0}
DECL FDAT FP111={TOOL_NO 1,BASE_NO 3,IPO_FRAME #BASE,POINT2[] " ",TQ_STATE FALSE}
DECL E6POS XP111={X 491.53075,Y -0.60207,Z 2105.79902,A 90,B 0,C 180,S 2,T 34,E1 0,E2 0,E3 0,E4 0,E5 0,E6 0}
; DECL LDAT LCPDATP2={VEL 1,ACC 100,APO_DIST 100,APO_FAC 50.0,ORI_TYP #VAR,CIRC_TYP #BASE,JERK_FAC 50.0}
DECL FDAT FP112={TOOL_NO 1,BASE_NO 3,IPO_FRAME #BASE,POINT2[] " ",TQ_STATE FALSE}
DECL E6POS XP112={X 491.53075,Y -0.6016,Z 1426.77049,A 90,B 0,C -180,S 2,T 34,E1 0,E2 0,E3 0,E4 0,E5 0,E6 0}
; DECL LDAT LCPDATP1={VEL 1,ACC 100,APO_DIST 100,APO_FAC 50.0,ORI_TYP #VAR,CIRC_TYP #BASE,JERK_FAC 50.0}
DECL FDAT FPick_E_1_P_3={TOOL_NO 1,BASE_NO 3,IPO_FRAME #BASE,POINT2[] " ",TQ_STATE FALSE}
DECL E6POS XPick_E_1_P_3={X 491.53075,Y 56.83161,Z 1343.55737,A 90,B 0,C -180,S 2,T 34,E1 0,E2 0,E3 0,E4 0,E5 0,E6 0}
; DECL LDAT LCPDATP3={VEL 1,ACC 100,APO_DIST 100,APO_FAC 50.0,ORI_TYP #VAR,CIRC_TYP #BASE,JERK_FAC 50.0}
DECL FDAT FP114={TOOL_NO 1,BASE_NO 3,IPO_FRAME #BASE,POINT2[] " ",TQ_STATE FALSE}
DECL E6POS XP114={X 491.53075,Y 56.83161,Z 2105.80057,A 90,B 0,C 180,S 2,T 34,E1 0,E2 0,E3 0,E4 0,E5 0,E6 0}
; ENDDAT for Pick_E_1_P_3
; Data for AbreGarraOp1
; ENDDAT for AbreGarraOp1
; Data for Pick_E_1_P_6
; DECL PDAT PPDATP1={VEL 100,ACC 100,APO_DIST 100,APO_MODE #CDIS,GEAR_JERK 100.000,EXAX_IGN 0}
DECL FDAT FP242={TOOL_NO 1,BASE_NO 3,IPO_FRAME #BASE,POINT2[] " ",TQ_STATE FALSE}
DECL E6POS XP242={X 549.54063,Y 572.77209,Z 2105.79938,A -90,B 0,C -180,S 2,T 2,E1 0,E2 0,E3 0,E4 0,E5 0,E6 0}
; DECL LDAT LCPDATP2={VEL 1,ACC 100,APO_DIST 100,APO_FAC 50.0,ORI_TYP #VAR,CIRC_TYP #BASE,JERK_FAC 50.0}
DECL FDAT FP243={TOOL_NO 1,BASE_NO 3,IPO_FRAME #BASE,POINT2[] " ",TQ_STATE FALSE}
DECL E6POS XP243={X 549.54041,Y 572.77209,Z 1426.77049,A -90,B 0,C -180,S 2,T 2,E1 0,E2 0,E3 0,E4 0,E5 0,E6 0}
; DECL LDAT LCPDATP1={VEL 1,ACC 100,APO_DIST 100,APO_FAC 50.0,ORI_TYP #VAR,CIRC_TYP #BASE,JERK_FAC 50.0}
DECL FDAT FPick_E_1_P_6={TOOL_NO 1,BASE_NO 3,IPO_FRAME #BASE,POINT2[] " ",TQ_STATE FALSE}
DECL E6POS XPick_E_1_P_6={X 549.54041,Y 651.48646,Z 1343.55737,A -90,B 0,C -180,S 2,T 2,E1 0,E2 0,E3 0,E4 0,E5 0,E6 0}
; DECL LDAT LCPDATP3={VEL 1,ACC 100,APO_DIST 100,APO_FAC 50.0,ORI_TYP #VAR,CIRC_TYP #BASE,JERK_FAC 50.0}
DECL FDAT FP245={TOOL_NO 1,BASE_NO 3,IPO_FRAME #BASE,POINT2[] " ",TQ_STATE FALSE}
DECL E6POS XP245={X 549.53996,Y 572.77209,Z 2105.80057,A -90,B 0,C 180,S 2,T 2,E1 0,E2 0,E3 0,E4 0,E5 0,E6 0}
; ENDDAT for Pick_E_1_P_6
; Data for Pick_E_1_P_4
; DECL PDAT PPDATP1={VEL 100,ACC 100,APO_DIST 100,APO_MODE #CDIS,GEAR_JERK 100.000,EXAX_IGN 0}
DECL FDAT FP391={TOOL_NO 1,BASE_NO 3,IPO_FRAME #BASE,POINT2[] " ",TQ_STATE FALSE}
DECL E6POS XP391={X 471.75075,Y 572.77234,Z 2105.79985,A -90,B 0,C -180,S 2,T 2,E1 0,E2 0,E3 0,E4 0,E5 0,E6 0}
; DECL LDAT LCPDATP2={VEL 1,ACC 100,APO_DIST 100,APO_FAC 50.0,ORI_TYP #VAR,CIRC_TYP #BASE,JERK_FAC 50.0}
DECL FDAT FP392={TOOL_NO 1,BASE_NO 3,IPO_FRAME #BASE,POINT2[] " ",TQ_STATE FALSE}
DECL E6POS XP392={X 471.75075,Y 572.77209,Z 1387.24782,A -90,B 0,C -180,S 2,T 2,E1 0,E2 0,E3 0,E4 0,E5 0,E6 0}
; DECL LDAT LCPDATP1={VEL 1,ACC 100,APO_DIST 100,APO_FAC 50.0,ORI_TYP #VAR,CIRC_TYP #BASE,JERK_FAC 50.0}
DECL FDAT FPick_E_1_P_4={TOOL_NO 1,BASE_NO 3,IPO_FRAME #BASE,POINT2[] " ",TQ_STATE FALSE}
DECL E6POS XPick_E_1_P_4={X 471.75075,Y 502.13363,Z 1392.47867,A -90,B 0,C -180,S 2,T 2,E1 0,E2 0,E3 0,E4 0,E5 0,E6 0}
; DECL LDAT LCPDATP3={VEL 1,ACC 100,APO_DIST 100,APO_FAC 50.0,ORI_TYP #VAR,CIRC_TYP #BASE,JERK_FAC 50.0}
DECL FDAT FP394={TOOL_NO 1,BASE_NO 3,IPO_FRAME #BASE,POINT2[] " ",TQ_STATE FALSE}
DECL E6POS XP394={X 471.75075,Y 502.13363,Z 2105.80057,A -90,B 0,C 180,S 2,T 2,E1 0,E2 0,E3 0,E4 0,E5 0,E6 0}
; ENDDAT for Pick_E_1_P_4
; Data for ConfGarraOp4
; ENDDAT for ConfGarraOp4
; Data for Pick_E_1_P_5
; DECL PDAT PPDATP1={VEL 100,ACC 100,APO_DIST 100,APO_MODE #CDIS,GEAR_JERK 100.000,EXAX_IGN 0}
DECL FDAT FP419={TOOL_NO 1,BASE_NO 3,IPO_FRAME #BASE,POINT2[] " ",TQ_STATE FALSE}
DECL E6POS XP419={X 489.59646,Y -2.83248,Z 2105.79954,A 90,B 0,C 180,S 2,T 34,E1 0,E2 0,E3 0,E4 0,E5 0,E6 0}
; DECL LDAT LCPDATP2={VEL 1,ACC 100,APO_DIST 100,APO_FAC 50.0,ORI_TYP #VAR,CIRC_TYP #BASE,JERK_FAC 50.0}
DECL FDAT FP424={TOOL_NO 1,BASE_NO 3,IPO_FRAME #BASE,POINT2[] " ",TQ_STATE FALSE}
DECL E6POS XP424={X 489.59646,Y -2.8321,Z 1392.47867,A 90,B 0,C -180,S 2,T 34,E1 0,E2 0,E3 0,E4 0,E5 0,E6 0}
; DECL LDAT LCPDATP1={VEL 1,ACC 100,APO_DIST 100,APO_FAC 50.0,ORI_TYP #VAR,CIRC_TYP #BASE,JERK_FAC 50.0}
DECL FDAT FPick_E_1_P_5={TOOL_NO 1,BASE_NO 3,IPO_FRAME #BASE,POINT2[] " ",TQ_STATE FALSE}
DECL E6POS XPick_E_1_P_5={X 489.59646,Y 19.40185,Z 1392.47867,A 90,B 0,C -180,S 2,T 34,E1 0,E2 0,E3 0,E4 0,E5 0,E6 0}
; DECL LDAT LCPDATP3={VEL 1,ACC 100,APO_DIST 100,APO_FAC 50.0,ORI_TYP #VAR,CIRC_TYP #BASE,JERK_FAC 50.0}
DECL FDAT FP426={TOOL_NO 1,BASE_NO 3,IPO_FRAME #BASE,POINT2[] " ",TQ_STATE FALSE}
DECL E6POS XP426={X 489.59646,Y 19.40185,Z 2105.80057,A 90,B 0,C 180,S 2,T 34,E1 0,E2 0,E3 0,E4 0,E5 0,E6 0}
; ENDDAT for Pick_E_1_P_5
; Data for Mtrz_P2_2Aero
; DECL PDAT PPDATP2={VEL 100,ACC 100,APO_DIST 100,APO_MODE #CDIS,GEAR_JERK 100.000,EXAX_IGN 0}
DECL FDAT FP420={TOOL_NO 1,BASE_NO 2,IPO_FRAME #BASE,POINT2[] " ",TQ_STATE FALSE}
DECL E6POS XP420={X 653.58499,Y -68.23916,Z 1114.55813,A -90,B 0,C 180,S 2,T 35,E1 0,E2 0,E3 0,E4 0,E5 0,E6 0}
; DECL LDAT LCPDATP4={VEL 1,ACC 100,APO_DIST 100,APO_FAC 50.0,ORI_TYP #VAR,CIRC_TYP #BASE,JERK_FAC 50.0}
DECL FDAT FP421={TOOL_NO 1,BASE_NO 2,IPO_FRAME #BASE,POINT2[] " ",TQ_STATE FALSE}
DECL E6POS XP421={X 653.58503,Y -68.23958,Z 914.55818,A -90,B 0,C 180,S 2,T 35,E1 0,E2 0,E3 0,E4 0,E5 0,E6 0}
; DECL LDAT LCPDATP5={VEL 1,ACC 100,APO_DIST 100,APO_FAC 50.0,ORI_TYP #VAR,CIRC_TYP #BASE,JERK_FAC 50.0}
DECL FDAT FP422={TOOL_NO 1,BASE_NO 2,IPO_FRAME #BASE,POINT2[] " ",TQ_STATE FALSE}
DECL E6POS XP422={X 653.58552,Y 31.76059,Z 814.55872,A -90,B 0,C 180,S 2,T 35,E1 0,E2 0,E3 0,E4 0,E5 0,E6 0}
; DECL PDAT PPDATP3={VEL 100,ACC 100,APO_DIST 100,APO_MODE #CDIS,GEAR_JERK 100.000,EXAX_IGN 0}
DECL FDAT FP423={TOOL_NO 1,BASE_NO 2,IPO_FRAME #BASE,POINT2[] " ",TQ_STATE FALSE}
DECL E6POS XP423={X 653.58549,Y -379.23915,Z 1114.55842,A -90,B 0,C 180,S 2,T 35,E1 0,E2 0,E3 0,E4 0,E5 0,E6 0}
; DECL LDAT LCPDATP6={VEL 1,ACC 100,APO_DIST 100,APO_FAC 50.0,ORI_TYP #VAR,CIRC_TYP #BASE,JERK_FAC 50.0}
DECL FDAT FP427={TOOL_NO 1,BASE_NO 2,IPO_FRAME #BASE,POINT2[] " ",TQ_STATE FALSE}
DECL E6POS XP427={X 653.58555,Y -379.23964,Z 914.55731,A -90,B 0,C 180,S 2,T 35,E1 0,E2 0,E3 0,E4 0,E5 0,E6 0}
; DECL LDAT LCPDATP7={VEL 1,ACC 100,APO_DIST 100,APO_FAC 50.0,ORI_TYP #VAR,CIRC_TYP #BASE,JERK_FAC 50.0}
DECL FDAT FP428={TOOL_NO 1,BASE_NO 2,IPO_FRAME #BASE,POINT2[] " ",TQ_STATE FALSE}
DECL E6POS XP428={X 653.58531,Y -279.23915,Z 814.55827,A -90,B 0,C 180,S 2,T 35,E1 0,E2 0,E3 0,E4 0,E5 0,E6 0}
; DECL PDAT PPDATP4={VEL 100,ACC 100,APO_DIST 100,APO_MODE #CDIS,GEAR_JERK 100.000,EXAX_IGN 0}
DECL FDAT FP429={TOOL_NO 1,BASE_NO 2,IPO_FRAME #BASE,POINT2[] " ",TQ_STATE FALSE}
DECL E6POS XP429={X 653.58596,Y -690.23907,Z 1114.55772,A -90,B 0,C 180,S 2,T 35,E1 0,E2 0,E3 0,E4 0,E5 0,E6 0}
; DECL LDAT LCPDATP8={VEL 1,ACC 100,APO_DIST 100,APO_FAC 50.0,ORI_TYP #VAR,CIRC_TYP #BASE,JERK_FAC 50.0}
DECL FDAT FP430={TOOL_NO 1,BASE_NO 2,IPO_FRAME #BASE,POINT2[] " ",TQ_STATE FALSE}
DECL E6POS XP430={X 653.58602,Y -690.23957,Z 914.55732,A -90,B 0,C 180,S 2,T 35,E1 0,E2 0,E3 0,E4 0,E5 0,E6 0}
; DECL LDAT LCPDATP9={VEL 1,ACC 100,APO_DIST 100,APO_FAC 50.0,ORI_TYP #VAR,CIRC_TYP #BASE,JERK_FAC 50.0}
DECL FDAT FP431={TOOL_NO 1,BASE_NO 2,IPO_FRAME #BASE,POINT2[] " ",TQ_STATE FALSE}
DECL E6POS XP431={X 653.58453,Y -590.23945,Z 814.55813,A -90,B 0,C 180,S 2,T 35,E1 0,E2 0,E3 0,E4 0,E5 0,E6 0}
; ENDDAT for Mtrz_P2_2Aero
; Data for Pick_E_2_P_1
; DECL PDAT PPDATP1={VEL 100,ACC 100,APO_DIST 100,APO_MODE #CDIS,GEAR_JERK 100.000,EXAX_IGN 0}
DECL FDAT FP441={TOOL_NO 1,BASE_NO 4,IPO_FRAME #BASE,POINT2[] " ",TQ_STATE FALSE}
DECL E6POS XP441={X 598.63538,Y 78.06412,Z 2072.81644,A -90,B 0,C -180,S 2,T 3,E1 0,E2 0,E3 0,E4 0,E5 0,E6 0}
; DECL LDAT LCPDATP2={VEL 1,ACC 100,APO_DIST 100,APO_FAC 50.0,ORI_TYP #VAR,CIRC_TYP #BASE,JERK_FAC 50.0}
DECL FDAT FP442={TOOL_NO 1,BASE_NO 4,IPO_FRAME #BASE,POINT2[] " ",TQ_STATE FALSE}
DECL E6POS XP442={X 598.63486,Y 78.06328,Z 1393.78838,A -90,B 0,C -180,S 2,T 3,E1 0,E2 0,E3 0,E4 0,E5 0,E6 0}
; DECL LDAT LCPDATP1={VEL 1,ACC 100,APO_DIST 100,APO_FAC 50.0,ORI_TYP #VAR,CIRC_TYP #BASE,JERK_FAC 50.0}
DECL FDAT FPick_E_2_P_1={TOOL_NO 1,BASE_NO 4,IPO_FRAME #BASE,POINT2[] " ",TQ_STATE FALSE}
DECL E6POS XPick_E_2_P_1={X 598.63515,Y 7.10195,Z 1343.57449,A -90,B 0,C 180,S 2,T 3,E1 0,E2 0,E3 0,E4 0,E5 0,E6 0}
; DECL LDAT LCPDATP3={VEL 1,ACC 100,APO_DIST 100,APO_FAC 50.0,ORI_TYP #VAR,CIRC_TYP #BASE,JERK_FAC 50.0}
DECL FDAT FP443={TOOL_NO 1,BASE_NO 4,IPO_FRAME #BASE,POINT2[] " ",TQ_STATE FALSE}
DECL E6POS XP443={X 598.635,Y 7.10171,Z 2072.81825,A -90,B 0,C -180,S 2,T 3,E1 0,E2 0,E3 0,E4 0,E5 0,E6 0}
; ENDDAT for Pick_E_2_P_1
; Data for Mtrz_P2_5Aero
; DECL PDAT PPDATP6={VEL 100,ACC 100,APO_DIST 100,APO_MODE #CDIS,GEAR_JERK 100.000,EXAX_IGN 0}
DECL FDAT FP444={TOOL_NO 1,BASE_NO 2,IPO_FRAME #BASE,POINT2[] " ",TQ_STATE FALSE}
DECL E6POS XP444={X 1100.19013,Y -617.6956,Z 1064.55966,A -180,B 0,C 180,S 2,T 35,E1 0,E2 0,E3 0,E4 0,E5 0,E6 0}
; DECL LDAT LCPDATP12={VEL 1,ACC 100,APO_DIST 100,APO_FAC 50.0,ORI_TYP #VAR,CIRC_TYP #BASE,JERK_FAC 50.0}
DECL FDAT FP445={TOOL_NO 1,BASE_NO 2,IPO_FRAME #BASE,POINT2[] " ",TQ_STATE FALSE}
DECL E6POS XP445={X 1100.19109,Y -617.69559,Z 914.55854,A -180,B 0,C 180,S 2,T 35,E1 0,E2 0,E3 0,E4 0,E5 0,E6 0}
; DECL LDAT LCPDATP11={VEL 1,ACC 100,APO_DIST 100,APO_FAC 50.0,ORI_TYP #VAR,CIRC_TYP #BASE,JERK_FAC 50.0}
DECL FDAT FP446={TOOL_NO 1,BASE_NO 2,IPO_FRAME #BASE,POINT2[] " ",TQ_STATE FALSE}
DECL E6POS XP446={X 1200.19026,Y -617.69557,Z 814.55914,A 180,B 0,C 180,S 2,T 35,E1 0,E2 0,E3 0,E4 0,E5 0,E6 0}
; DECL PDAT PPDATP7={VEL 100,ACC 100,APO_DIST 100,APO_MODE #CDIS,GEAR_JERK 100.000,EXAX_IGN 0}
DECL FDAT FP447={TOOL_NO 1,BASE_NO 2,IPO_FRAME #BASE,POINT2[] " ",TQ_STATE FALSE}
DECL E6POS XP447={X 740.1904,Y -617.69575,Z 1064.55904,A 180,B 0,C -180,S 2,T 35,E1 0,E2 0,E3 0,E4 0,E5 0,E6 0}
; DECL LDAT LCPDATP13={VEL 1,ACC 100,APO_DIST 100,APO_FAC 50.0,ORI_TYP #VAR,CIRC_TYP #BASE,JERK_FAC 50.0}
DECL FDAT FP448={TOOL_NO 1,BASE_NO 2,IPO_FRAME #BASE,POINT2[] " ",TQ_STATE FALSE}
DECL E6POS XP448={X 740.19091,Y -617.69576,Z 914.55853,A 180,B 0,C -180,S 2,T 35,E1 0,E2 0,E3 0,E4 0,E5 0,E6 0}
; DECL LDAT LCPDATP14={VEL 1,ACC 100,APO_DIST 100,APO_FAC 50.0,ORI_TYP #VAR,CIRC_TYP #BASE,JERK_FAC 50.0}
DECL FDAT FP449={TOOL_NO 1,BASE_NO 2,IPO_FRAME #BASE,POINT2[] " ",TQ_STATE FALSE}
DECL E6POS XP449={X 840.19068,Y -617.69567,Z 814.55885,A 180,B 0,C 180,S 2,T 35,E1 0,E2 0,E3 0,E4 0,E5 0,E6 0}
; DECL PDAT PPDATP8={VEL 100,ACC 100,APO_DIST 100,APO_MODE #CDIS,GEAR_JERK 100.000,EXAX_IGN 0}
DECL FDAT FP450={TOOL_NO 1,BASE_NO 2,IPO_FRAME #BASE,POINT2[] " ",TQ_STATE FALSE}
DECL E6POS XP450={X 380.19008,Y -617.69565,Z 1064.55907,A 180,B 0,C -180,S 2,T 35,E1 0,E2 0,E3 0,E4 0,E5 0,E6 0}
; DECL LDAT LCPDATP15={VEL 1,ACC 100,APO_DIST 100,APO_FAC 50.0,ORI_TYP #VAR,CIRC_TYP #BASE,JERK_FAC 50.0}
DECL FDAT FP451={TOOL_NO 1,BASE_NO 2,IPO_FRAME #BASE,POINT2[] " ",TQ_STATE FALSE}
DECL E6POS XP451={X 380.1905,Y -617.69547,Z 914.5591,A -180,B 0,C 180,S 2,T 35,E1 0,E2 0,E3 0,E4 0,E5 0,E6 0}
; DECL LDAT LCPDATP16={VEL 1,ACC 100,APO_DIST 100,APO_FAC 50.0,ORI_TYP #VAR,CIRC_TYP #BASE,JERK_FAC 50.0}
DECL FDAT FP452={TOOL_NO 1,BASE_NO 2,IPO_FRAME #BASE,POINT2[] " ",TQ_STATE FALSE}
DECL E6POS XP452={X 480.1904,Y -617.69581,Z 814.55931,A -180,B 0,C -180,S 2,T 35,E1 0,E2 0,E3 0,E4 0,E5 0,E6 0}
; ENDDAT for Mtrz_P2_5Aero
; Data for Mtrz_P2_17KitKat
; DECL PDAT PPDATP12={VEL 100,ACC 100,APO_DIST 100,APO_MODE #CDIS,GEAR_JERK 100.000,EXAX_IGN 0}
DECL FDAT FP462={TOOL_NO 1,BASE_NO 2,IPO_FRAME #BASE,POINT2[] " ",TQ_STATE FALSE}
DECL E6POS XP462={X 1164.97133,Y -659.2018,Z 1114.58702,A -180,B 0,C 180,S 2,T 35,E1 0,E2 0,E3 0,E4 0,E5 0,E6 0}
; DECL LDAT LCPDATP22={VEL 1,ACC 100,APO_DIST 100,APO_FAC 50.0,ORI_TYP #VAR,CIRC_TYP #BASE,JERK_FAC 50.0}
DECL FDAT FP463={TOOL_NO 1,BASE_NO 2,IPO_FRAME #BASE,POINT2[] " ",TQ_STATE FALSE}
DECL E6POS XP463={X 1164.97124,Y -659.20201,Z 964.58697,A 180,B 0,C 180,S 2,T 35,E1 0,E2 0,E3 0,E4 0,E5 0,E6 0}
; DECL LDAT LCPDATP23={VEL 1,ACC 100,APO_DIST 100,APO_FAC 50.0,ORI_TYP #VAR,CIRC_TYP #BASE,JERK_FAC 50.0}
DECL FDAT FP464={TOOL_NO 1,BASE_NO 2,IPO_FRAME #BASE,POINT2[] " ",TQ_STATE FALSE}
DECL E6POS XP464={X 1264.97156,Y -659.2018,Z 814.58693,A 180,B 0,C -180,S 2,T 35,E1 0,E2 0,E3 0,E4 0,E5 0,E6 0}
; DECL PDAT PPDATP13={VEL 100,ACC 100,APO_DIST 100,APO_MODE #CDIS,GEAR_JERK 100.000,EXAX_IGN 0}
DECL FDAT FP465={TOOL_NO 1,BASE_NO 2,IPO_FRAME #BASE,POINT2[] " ",TQ_STATE FALSE}
DECL E6POS XP465={X 864.97209,Y -659.20155,Z 1114.58693,A -180,B 0,C 180,S 2,T 35,E1 0,E2 0,E3 0,E4 0,E5 0,E6 0}
; DECL LDAT LCPDATP24={VEL 1,ACC 100,APO_DIST 100,APO_FAC 50.0,ORI_TYP #VAR,CIRC_TYP #BASE,JERK_FAC 50.0}
DECL FDAT FP466={TOOL_NO 1,BASE_NO 2,IPO_FRAME #BASE,POINT2[] " ",TQ_STATE FALSE}
DECL E6POS XP466={X 864.97244,Y -659.20212,Z 964.58694,A 180,B 0,C -180,S 2,T 35,E1 0,E2 0,E3 0,E4 0,E5 0,E6 0}
; DECL LDAT LCPDATP25={VEL 1,ACC 100,APO_DIST 100,APO_FAC 50.0,ORI_TYP #VAR,CIRC_TYP #BASE,JERK_FAC 50.0}
DECL FDAT FP467={TOOL_NO 1,BASE_NO 2,IPO_FRAME #BASE,POINT2[] " ",TQ_STATE FALSE}
DECL E6POS XP467={X 964.97194,Y -659.20202,Z 814.58663,A 180,B 0,C 180,S 2,T 35,E1 0,E2 0,E3 0,E4 0,E5 0,E6 0}
; DECL PDAT PPDATP14={VEL 100,ACC 100,APO_DIST 100,APO_MODE #CDIS,GEAR_JERK 100.000,EXAX_IGN 0}
DECL FDAT FP468={TOOL_NO 1,BASE_NO 2,IPO_FRAME #BASE,POINT2[] " ",TQ_STATE FALSE}
DECL E6POS XP468={X 564.97227,Y -659.20224,Z 1114.58651,A -180,B 0,C 180,S 2,T 35,E1 0,E2 0,E3 0,E4 0,E5 0,E6 0}
; DECL LDAT LCPDATP26={VEL 1,ACC 100,APO_DIST 100,APO_FAC 50.0,ORI_TYP #VAR,CIRC_TYP #BASE,JERK_FAC 50.0}
DECL FDAT FP469={TOOL_NO 1,BASE_NO 2,IPO_FRAME #BASE,POINT2[] " ",TQ_STATE FALSE}
DECL E6POS XP469={X 564.97232,Y -659.20204,Z 964.58683,A -180,B 0,C -180,S 2,T 35,E1 0,E2 0,E3 0,E4 0,E5 0,E6 0}
; DECL LDAT LCPDATP27={VEL 1,ACC 100,APO_DIST 100,APO_FAC 50.0,ORI_TYP #VAR,CIRC_TYP #BASE,JERK_FAC 50.0}
DECL FDAT FP470={TOOL_NO 1,BASE_NO 2,IPO_FRAME #BASE,POINT2[] " ",TQ_STATE FALSE}
DECL E6POS XP470={X 664.97218,Y -659.20207,Z 814.5867,A 180,B 0,C -180,S 2,T 35,E1 0,E2 0,E3 0,E4 0,E5 0,E6 0}
; DECL PDAT PPDATP15={VEL 100,ACC 100,APO_DIST 100,APO_MODE #CDIS,GEAR_JERK 100.000,EXAX_IGN 0}
DECL FDAT FP471={TOOL_NO 1,BASE_NO 2,IPO_FRAME #BASE,POINT2[] " ",TQ_STATE FALSE}
DECL E6POS XP471={X 314.97186,Y -659.20226,Z 1114.58777,A -180,B 0,C -180,S 2,T 35,E1 0,E2 0,E3 0,E4 0,E5 0,E6 0}
; DECL LDAT LCPDATP29={VEL 1,ACC 100,APO_DIST 100,APO_FAC 50.0,ORI_TYP #VAR,CIRC_TYP #BASE,JERK_FAC 50.0}
DECL FDAT FP472={TOOL_NO 1,BASE_NO 2,IPO_FRAME #BASE,POINT2[] " ",TQ_STATE FALSE}
DECL E6POS XP472={X 314.97221,Y -659.202,Z 964.5866,A 180,B 0,C -180,S 2,T 35,E1 0,E2 0,E3 0,E4 0,E5 0,E6 0}
; DECL LDAT LCPDATP28={VEL 1,ACC 100,APO_DIST 100,APO_FAC 50.0,ORI_TYP #VAR,CIRC_TYP #BASE,JERK_FAC 50.0}
DECL FDAT FP473={TOOL_NO 1,BASE_NO 2,IPO_FRAME #BASE,POINT2[] " ",TQ_STATE FALSE}
DECL E6POS XP473={X 364.97196,Y -659.20185,Z 814.58667,A -180,B 0,C 180,S 2,T 35,E1 0,E2 0,E3 0,E4 0,E5 0,E6 0}
; ENDDAT for Mtrz_P2_17KitKat
; Data for Mtrz_P2_20KitKat
; DECL PDAT PPDATP39={VEL 100,ACC 100,APO_DIST 100,APO_MODE #CDIS,GEAR_JERK 100.000,EXAX_IGN 0}
DECL FDAT FP486={TOOL_NO 1,BASE_NO 2,IPO_FRAME #BASE,POINT2[] " ",TQ_STATE FALSE}
DECL E6POS XP486={X 631.89876,Y -60.28636,Z 984.57724,A -90,B 0,C 180,S 2,T 35,E1 0,E2 0,E3 0,E4 0,E5 0,E6 0}
; DECL LDAT LCPDATP76={VEL 1,ACC 100,APO_DIST 100,APO_FAC 50.0,ORI_TYP #VAR,CIRC_TYP #BASE,JERK_FAC 50.0}
DECL FDAT FP487={TOOL_NO 1,BASE_NO 2,IPO_FRAME #BASE,POINT2[] " ",TQ_STATE FALSE}
DECL E6POS XP487={X 631.89872,Y -60.28599,Z 864.5794,A -90,B 0,C 180,S 2,T 35,E1 0,E2 0,E3 0,E4 0,E5 0,E6 0}
; DECL LDAT LCPDATP87={VEL 1,ACC 100,APO_DIST 100,APO_FAC 50.0,ORI_TYP #VAR,CIRC_TYP #BASE,JERK_FAC 50.0}
DECL FDAT FP488={TOOL_NO 1,BASE_NO 2,IPO_FRAME #BASE,POINT2[] " ",TQ_STATE FALSE}
DECL E6POS XP488={X 631.89823,Y 39.71353,Z 814.57776,A -90,B 0,C 180,S 2,T 35,E1 0,E2 0,E3 0,E4 0,E5 0,E6 0}
; DECL PDAT PPDATP45={VEL 100,ACC 100,APO_DIST 100,APO_MODE #CDIS,GEAR_JERK 100.000,EXAX_IGN 0}
DECL FDAT FP489={TOOL_NO 1,BASE_NO 2,IPO_FRAME #BASE,POINT2[] " ",TQ_STATE FALSE}
DECL E6POS XP489={X 631.91587,Y -326.28876,Z 984.57652,A -90,B 0,C 180,S 2,T 35,E1 0,E2 0,E3 0,E4 0,E5 0,E6 0}
; DECL LDAT LCPDATP88={VEL 1,ACC 100,APO_DIST 100,APO_FAC 50.0,ORI_TYP #VAR,CIRC_TYP #BASE,JERK_FAC 50.0}
DECL FDAT FP490={TOOL_NO 1,BASE_NO 2,IPO_FRAME #BASE,POINT2[] " ",TQ_STATE FALSE}
DECL E6POS XP490={X 631.9158,Y -326.2882,Z 864.57941,A -90,B 0,C 180,S 2,T 35,E1 0,E2 0,E3 0,E4 0,E5 0,E6 0}
; DECL LDAT LCPDATP89={VEL 1,ACC 100,APO_DIST 100,APO_FAC 50.0,ORI_TYP #VAR,CIRC_TYP #BASE,JERK_FAC 50.0}
DECL FDAT FP491={TOOL_NO 1,BASE_NO 2,IPO_FRAME #BASE,POINT2[] " ",TQ_STATE FALSE}
DECL E6POS XP491={X 631.91592,Y -276.28848,Z 814.57799,A -90,B 0,C 180,S 2,T 35,E1 0,E2 0,E3 0,E4 0,E5 0,E6 0}
; DECL PDAT PPDATP46={VEL 100,ACC 100,APO_DIST 100,APO_MODE #CDIS,GEAR_JERK 100.000,EXAX_IGN 0}
DECL FDAT FP492={TOOL_NO 1,BASE_NO 2,IPO_FRAME #BASE,POINT2[] " ",TQ_STATE FALSE}
DECL E6POS XP492={X 631.8987,Y -642.28053,Z 984.57749,A -90,B 0,C 180,S 2,T 35,E1 0,E2 0,E3 0,E4 0,E5 0,E6 0}
; DECL LDAT LCPDATP91={VEL 1,ACC 100,APO_DIST 100,APO_FAC 50.0,ORI_TYP #VAR,CIRC_TYP #BASE,JERK_FAC 50.0}
DECL FDAT FP493={TOOL_NO 1,BASE_NO 2,IPO_FRAME #BASE,POINT2[] " ",TQ_STATE FALSE}
DECL E6POS XP493={X 631.89872,Y -642.28071,Z 864.57933,A -90,B 0,C 180,S 2,T 35,E1 0,E2 0,E3 0,E4 0,E5 0,E6 0}
; DECL LDAT LCPDATP90={VEL 1,ACC 100,APO_DIST 100,APO_FAC 50.0,ORI_TYP #VAR,CIRC_TYP #BASE,JERK_FAC 50.0}
DECL FDAT FP494={TOOL_NO 1,BASE_NO 2,IPO_FRAME #BASE,POINT2[] " ",TQ_STATE FALSE}
DECL E6POS XP494={X 631.89799,Y -592.28052,Z 814.57699,A -90,B 0,C 180,S 2,T 35,E1 0,E2 0,E3 0,E4 0,E5 0,E6 0}
; ENDDAT for Mtrz_P2_20KitKat
; Data for Mtrz_P2_11CoffeCrisp
; DECL PDAT PPDATP16={VEL 100,ACC 100,APO_DIST 100,APO_MODE #CDIS,GEAR_JERK 100.000,EXAX_IGN 0}
DECL FDAT FP495={TOOL_NO 1,BASE_NO 2,IPO_FRAME #BASE,POINT2[] " ",TQ_STATE FALSE}
DECL E6POS XP495={X 1151.36786,Y -631.42176,Z 1064.5494,A -180,B 0,C 180,S 2,T 35,E1 0,E2 0,E3 0,E4 0,E5 0,E6 0}
; DECL LDAT LCPDATP30={VEL 1,ACC 100,APO_DIST 100,APO_FAC 50.0,ORI_TYP #VAR,CIRC_TYP #BASE,JERK_FAC 50.0}
DECL FDAT FP496={TOOL_NO 1,BASE_NO 2,IPO_FRAME #BASE,POINT2[] " ",TQ_STATE FALSE}
DECL E6POS XP496={X 1151.36819,Y -631.42194,Z 964.54979,A 180,B 0,C -180,S 2,T 35,E1 0,E2 0,E3 0,E4 0,E5 0,E6 0}
; DECL LDAT LCPDATP31={VEL 1,ACC 100,APO_DIST 100,APO_FAC 50.0,ORI_TYP #VAR,CIRC_TYP #BASE,JERK_FAC 50.0}
DECL FDAT FP497={TOOL_NO 1,BASE_NO 2,IPO_FRAME #BASE,POINT2[] " ",TQ_STATE FALSE}
DECL E6POS XP497={X 1251.36773,Y -631.42178,Z 814.55016,A 180,B 0,C -180,S 2,T 35,E1 0,E2 0,E3 0,E4 0,E5 0,E6 0}
; DECL PDAT PPDATP17={VEL 100,ACC 100,APO_DIST 100,APO_MODE #CDIS,GEAR_JERK 100.000,EXAX_IGN 0}
DECL FDAT FP498={TOOL_NO 1,BASE_NO 2,IPO_FRAME #BASE,POINT2[] " ",TQ_STATE FALSE}
DECL E6POS XP498={X 757.36759,Y -631.42217,Z 1064.55065,A -180,B 0,C 180,S 2,T 35,E1 0,E2 0,E3 0,E4 0,E5 0,E6 0}
; DECL LDAT LCPDATP32={VEL 1,ACC 100,APO_DIST 100,APO_FAC 50.0,ORI_TYP #VAR,CIRC_TYP #BASE,JERK_FAC 50.0}
DECL FDAT FP499={TOOL_NO 1,BASE_NO 2,IPO_FRAME #BASE,POINT2[] " ",TQ_STATE FALSE}
DECL E6POS XP499={X 757.36707,Y -631.42216,Z 964.55002,A 180,B 0,C 180,S 2,T 35,E1 0,E2 0,E3 0,E4 0,E5 0,E6 0}
; DECL LDAT LCPDATP33={VEL 1,ACC 100,APO_DIST 100,APO_FAC 50.0,ORI_TYP #VAR,CIRC_TYP #BASE,JERK_FAC 50.0}
DECL FDAT FP500={TOOL_NO 1,BASE_NO 2,IPO_FRAME #BASE,POINT2[] " ",TQ_STATE FALSE}
DECL E6POS XP500={X 857.36783,Y -631.42166,Z 814.55037,A 180,B 0,C -180,S 2,T 35,E1 0,E2 0,E3 0,E4 0,E5 0,E6 0}
; DECL PDAT PPDATP18={VEL 100,ACC 100,APO_DIST 100,APO_MODE #CDIS,GEAR_JERK 100.000,EXAX_IGN 0}
DECL FDAT FP501={TOOL_NO 1,BASE_NO 2,IPO_FRAME #BASE,POINT2[] " ",TQ_STATE FALSE}
DECL E6POS XP501={X 363.36782,Y -631.42184,Z 1064.54989,A -180,B 0,C 180,S 2,T 35,E1 0,E2 0,E3 0,E4 0,E5 0,E6 0}
; DECL LDAT LCPDATP34={VEL 1,ACC 100,APO_DIST 100,APO_FAC 50.0,ORI_TYP #VAR,CIRC_TYP #BASE,JERK_FAC 50.0}
DECL FDAT FP502={TOOL_NO 1,BASE_NO 2,IPO_FRAME #BASE,POINT2[] " ",TQ_STATE FALSE}
DECL E6POS XP502={X 363.36773,Y -631.42215,Z 964.55039,A 180,B 0,C -180,S 2,T 35,E1 0,E2 0,E3 0,E4 0,E5 0,E6 0}
; DECL LDAT LCPDATP35={VEL 1,ACC 100,APO_DIST 100,APO_FAC 50.0,ORI_TYP #VAR,CIRC_TYP #BASE,JERK_FAC 50.0}
DECL FDAT FP503={TOOL_NO 1,BASE_NO 2,IPO_FRAME #BASE,POINT2[] " ",TQ_STATE FALSE}
DECL E6POS XP503={X 463.36751,Y -631.42168,Z 814.54997,A 180,B 0,C 180,S 2,T 35,E1 0,E2 0,E3 0,E4 0,E5 0,E6 0}
; ENDDAT for Mtrz_P2_11CoffeCrisp
; Data for Mtrz_P2_21KitKat
; DECL PDAT PPDATP9={VEL 100,ACC 100,APO_DIST 100,APO_MODE #CDIS,GEAR_JERK 100.000,EXAX_IGN 0}
DECL FDAT FP513={TOOL_NO 1,BASE_NO 2,IPO_FRAME #BASE,POINT2[] " ",TQ_STATE FALSE}
DECL E6POS XP513={X 660.98163,Y -70.79127,Z 1064.5138,A -90,B 0,C 180,S 2,T 35,E1 0,E2 0,E3 0,E4 0,E5 0,E6 0}
; DECL LDAT LCPDATP10={VEL 1,ACC 100,APO_DIST 100,APO_FAC 50.0,ORI_TYP #VAR,CIRC_TYP #BASE,JERK_FAC 50.0}
DECL FDAT FP514={TOOL_NO 1,BASE_NO 2,IPO_FRAME #BASE,POINT2[] " ",TQ_STATE FALSE}
DECL E6POS XP514={X 660.98165,Y -70.79145,Z 964.51414,A -90,B 0,C 180,S 2,T 35,E1 0,E2 0,E3 0,E4 0,E5 0,E6 0}
; DECL LDAT LCPDATP17={VEL 1,ACC 100,APO_DIST 100,APO_FAC 50.0,ORI_TYP #VAR,CIRC_TYP #BASE,JERK_FAC 50.0}
DECL FDAT FP515={TOOL_NO 1,BASE_NO 2,IPO_FRAME #BASE,POINT2[] " ",TQ_STATE FALSE}
DECL E6POS XP515={X 660.98189,Y 29.20866,Z 814.51421,A -90,B 0,C 180,S 2,T 35,E1 0,E2 0,E3 0,E4 0,E5 0,E6 0}
; DECL PDAT PPDATP10={VEL 100,ACC 100,APO_DIST 100,APO_MODE #CDIS,GEAR_JERK 100.000,EXAX_IGN 0}
DECL FDAT FP516={TOOL_NO 1,BASE_NO 2,IPO_FRAME #BASE,POINT2[] " ",TQ_STATE FALSE}
DECL E6POS XP516={X 660.9826,Y -380.79111,Z 1064.51482,A -90,B 0,C 180,S 2,T 35,E1 0,E2 0,E3 0,E4 0,E5 0,E6 0}
; DECL LDAT LCPDATP18={VEL 1,ACC 100,APO_DIST 100,APO_FAC 50.0,ORI_TYP #VAR,CIRC_TYP #BASE,JERK_FAC 50.0}
DECL FDAT FP517={TOOL_NO 1,BASE_NO 2,IPO_FRAME #BASE,POINT2[] " ",TQ_STATE FALSE}
DECL E6POS XP517={X 660.98261,Y -380.7912,Z 964.51426,A -90,B 0,C 180,S 2,T 35,E1 0,E2 0,E3 0,E4 0,E5 0,E6 0}
; DECL LDAT LCPDATP19={VEL 1,ACC 100,APO_DIST 100,APO_FAC 50.0,ORI_TYP #VAR,CIRC_TYP #BASE,JERK_FAC 50.0}
DECL FDAT FP518={TOOL_NO 1,BASE_NO 2,IPO_FRAME #BASE,POINT2[] " ",TQ_STATE FALSE}
DECL E6POS XP518={X 660.98162,Y -280.79183,Z 814.51402,A -90,B 0,C 180,S 2,T 35,E1 0,E2 0,E3 0,E4 0,E5 0,E6 0}
; DECL PDAT PPDATP11={VEL 100,ACC 100,APO_DIST 100,APO_MODE #CDIS,GEAR_JERK 100.000,EXAX_IGN 0}
DECL FDAT FP519={TOOL_NO 1,BASE_NO 2,IPO_FRAME #BASE,POINT2[] " ",TQ_STATE FALSE}
DECL E6POS XP519={X 660.98221,Y -690.79115,Z 1064.51435,A -90,B 0,C 180,S 2,T 35,E1 0,E2 0,E3 0,E4 0,E5 0,E6 0}
; DECL LDAT LCPDATP20={VEL 1,ACC 100,APO_DIST 100,APO_FAC 50.0,ORI_TYP #VAR,CIRC_TYP #BASE,JERK_FAC 50.0}
DECL FDAT FP520={TOOL_NO 1,BASE_NO 2,IPO_FRAME #BASE,POINT2[] " ",TQ_STATE FALSE}
DECL E6POS XP520={X 660.98222,Y -690.79122,Z 964.51373,A -90,B 0,C 180,S 2,T 35,E1 0,E2 0,E3 0,E4 0,E5 0,E6 0}
; DECL LDAT LCPDATP21={VEL 1,ACC 100,APO_DIST 100,APO_FAC 50.0,ORI_TYP #VAR,CIRC_TYP #BASE,JERK_FAC 50.0}
DECL FDAT FP521={TOOL_NO 1,BASE_NO 2,IPO_FRAME #BASE,POINT2[] " ",TQ_STATE FALSE}
DECL E6POS XP521={X 660.98187,Y -590.791,Z 814.51382,A -90,B 0,C 180,S 2,T 35,E1 0,E2 0,E3 0,E4 0,E5 0,E6 0}
; ENDDAT for Mtrz_P2_21KitKat
; Data for Mtrz_P2_30All
; DECL PDAT PPDATP28={VEL 100,ACC 100,APO_DIST 100,APO_MODE #CDIS,GEAR_JERK 100.000,EXAX_IGN 0}
DECL FDAT FP522={TOOL_NO 1,BASE_NO 2,IPO_FRAME #BASE,POINT2[] " ",TQ_STATE FALSE}
DECL E6POS XP522={X 1121.61955,Y -600.37581,Z 1014.58069,A -180,B 0,C 180,S 2,T 35,E1 0,E2 0,E3 0,E4 0,E5 0,E6 0}
; DECL LDAT LCPDATP56={VEL 1,ACC 100,APO_DIST 100,APO_FAC 50.0,ORI_TYP #VAR,CIRC_TYP #BASE,JERK_FAC 50.0}
DECL FDAT FP523={TOOL_NO 1,BASE_NO 2,IPO_FRAME #BASE,POINT2[] " ",TQ_STATE FALSE}
DECL E6POS XP523={X 1121.61952,Y -600.37565,Z 914.58052,A -180,B 0,C 180,S 2,T 35,E1 0,E2 0,E3 0,E4 0,E5 0,E6 0}
; DECL LDAT LCPDATP57={VEL 1,ACC 100,APO_DIST 100,APO_FAC 50.0,ORI_TYP #VAR,CIRC_TYP #BASE,JERK_FAC 50.0}
DECL FDAT FP524={TOOL_NO 1,BASE_NO 2,IPO_FRAME #BASE,POINT2[] " ",TQ_STATE FALSE}
DECL E6POS XP524={X 1221.62029,Y -600.37588,Z 814.58116,A -180,B 0,C 180,S 2,T 35,E1 0,E2 0,E3 0,E4 0,E5 0,E6 0}
; DECL PDAT PPDATP30={VEL 100,ACC 100,APO_DIST 100,APO_MODE #CDIS,GEAR_JERK 100.000,EXAX_IGN 0}
DECL FDAT FP525={TOOL_NO 1,BASE_NO 2,IPO_FRAME #BASE,POINT2[] " ",TQ_STATE FALSE}
DECL E6POS XP525={X 841.61844,Y -600.37582,Z 1014.58086,A -180,B 0,C 180,S 2,T 35,E1 0,E2 0,E3 0,E4 0,E5 0,E6 0}
; DECL LDAT LCPDATP58={VEL 1,ACC 100,APO_DIST 100,APO_FAC 50.0,ORI_TYP #VAR,CIRC_TYP #BASE,JERK_FAC 50.0}
DECL FDAT FP526={TOOL_NO 1,BASE_NO 2,IPO_FRAME #BASE,POINT2[] " ",TQ_STATE FALSE}
DECL E6POS XP526={X 841.61889,Y -600.37591,Z 914.5811,A -180,B 0,C 180,S 2,T 35,E1 0,E2 0,E3 0,E4 0,E5 0,E6 0}
; DECL LDAT LCPDATP59={VEL 1,ACC 100,APO_DIST 100,APO_FAC 50.0,ORI_TYP #VAR,CIRC_TYP #BASE,JERK_FAC 50.0}
DECL FDAT FP527={TOOL_NO 1,BASE_NO 2,IPO_FRAME #BASE,POINT2[] " ",TQ_STATE FALSE}
DECL E6POS XP527={X 941.61934,Y -600.37549,Z 814.58096,A -180,B 0,C 180,S 2,T 35,E1 0,E2 0,E3 0,E4 0,E5 0,E6 0}
; DECL PDAT PPDATP31={VEL 100,ACC 100,APO_DIST 100,APO_MODE #CDIS,GEAR_JERK 100.000,EXAX_IGN 0}
DECL FDAT FP528={TOOL_NO 1,BASE_NO 2,IPO_FRAME #BASE,POINT2[] " ",TQ_STATE FALSE}
DECL E6POS XP528={X 561.61963,Y -600.3759,Z 1014.58096,A -180,B 0,C 180,S 2,T 35,E1 0,E2 0,E3 0,E4 0,E5 0,E6 0}
; DECL LDAT LCPDATP60={VEL 1,ACC 100,APO_DIST 100,APO_FAC 50.0,ORI_TYP #VAR,CIRC_TYP #BASE,JERK_FAC 50.0}
DECL FDAT FP529={TOOL_NO 1,BASE_NO 2,IPO_FRAME #BASE,POINT2[] " ",TQ_STATE FALSE}
DECL E6POS XP529={X 561.61982,Y -600.37581,Z 914.58075,A -180,B 0,C -180,S 2,T 35,E1 0,E2 0,E3 0,E4 0,E5 0,E6 0}
; DECL LDAT LCPDATP61={VEL 1,ACC 100,APO_DIST 100,APO_FAC 50.0,ORI_TYP #VAR,CIRC_TYP #BASE,JERK_FAC 50.0}
DECL FDAT FP530={TOOL_NO 1,BASE_NO 2,IPO_FRAME #BASE,POINT2[] " ",TQ_STATE FALSE}
DECL E6POS XP530={X 661.61919,Y -600.37586,Z 814.58067,A -180,B 0,C 180,S 2,T 35,E1 0,E2 0,E3 0,E4 0,E5 0,E6 0}
; DECL PDAT PPDATP32={VEL 100,ACC 100,APO_DIST 100,APO_MODE #CDIS,GEAR_JERK 100.000,EXAX_IGN 0}
DECL FDAT FP531={TOOL_NO 1,BASE_NO 2,IPO_FRAME #BASE,POINT2[] " ",TQ_STATE FALSE}
DECL E6POS XP531={X 331.61981,Y -600.37629,Z 1014.58119,A -180,B 0,C 180,S 2,T 35,E1 0,E2 0,E3 0,E4 0,E5 0,E6 0}
; DECL LDAT LCPDATP62={VEL 1,ACC 100,APO_DIST 100,APO_FAC 50.0,ORI_TYP #VAR,CIRC_TYP #BASE,JERK_FAC 50.0}
DECL FDAT FP532={TOOL_NO 1,BASE_NO 2,IPO_FRAME #BASE,POINT2[] " ",TQ_STATE FALSE}
DECL E6POS XP532={X 331.61926,Y -600.37595,Z 914.58081,A -180,B 0,C 180,S 2,T 35,E1 0,E2 0,E3 0,E4 0,E5 0,E6 0}
; DECL LDAT LCPDATP63={VEL 1,ACC 100,APO_DIST 100,APO_FAC 50.0,ORI_TYP #VAR,CIRC_TYP #BASE,JERK_FAC 50.0}
DECL FDAT FP533={TOOL_NO 1,BASE_NO 2,IPO_FRAME #BASE,POINT2[] " ",TQ_STATE FALSE}
DECL E6POS XP533={X 381.61985,Y -600.37563,Z 814.58067,A -180,B 0,C 180,S 2,T 35,E1 0,E2 0,E3 0,E4 0,E5 0,E6 0}
; ENDDAT for Mtrz_P2_30All
; Data for Mtrz_P2_24a28All
; DECL PDAT PPDATP33={VEL 100,ACC 100,APO_DIST 100,APO_MODE #CDIS,GEAR_JERK 100.000,EXAX_IGN 0}
DECL FDAT FP546={TOOL_NO 1,BASE_NO 2,IPO_FRAME #BASE,POINT2[] " ",TQ_STATE FALSE}
DECL E6POS XP546={X 598.506,Y -75.16847,Z 1014.54353,A -90,B 0,C 180,S 2,T 35,E1 0,E2 0,E3 0,E4 0,E5 0,E6 0}
; DECL LDAT LCPDATP64={VEL 1,ACC 100,APO_DIST 100,APO_FAC 50.0,ORI_TYP #VAR,CIRC_TYP #BASE,JERK_FAC 50.0}
DECL FDAT FP547={TOOL_NO 1,BASE_NO 2,IPO_FRAME #BASE,POINT2[] " ",TQ_STATE FALSE}
DECL E6POS XP547={X 598.50597,Y -75.1683,Z 914.54395,A -90,B 0,C 180,S 2,T 35,E1 0,E2 0,E3 0,E4 0,E5 0,E6 0}
; DECL LDAT LCPDATP65={VEL 1,ACC 100,APO_DIST 100,APO_FAC 50.0,ORI_TYP #VAR,CIRC_TYP #BASE,JERK_FAC 50.0}
DECL FDAT FP548={TOOL_NO 1,BASE_NO 2,IPO_FRAME #BASE,POINT2[] " ",TQ_STATE FALSE}
DECL E6POS XP548={X 598.50622,Y 24.83142,Z 814.54457,A -90,B 0,C 180,S 2,T 35,E1 0,E2 0,E3 0,E4 0,E5 0,E6 0}
; DECL PDAT PPDATP34={VEL 100,ACC 100,APO_DIST 100,APO_MODE #CDIS,GEAR_JERK 100.000,EXAX_IGN 0}
DECL FDAT FP549={TOOL_NO 1,BASE_NO 2,IPO_FRAME #BASE,POINT2[] " ",TQ_STATE FALSE}
DECL E6POS XP549={X 598.50633,Y -380.168,Z 1014.54476,A -90,B 0,C 180,S 2,T 35,E1 0,E2 0,E3 0,E4 0,E5 0,E6 0}
; DECL LDAT LCPDATP66={VEL 1,ACC 100,APO_DIST 100,APO_FAC 50.0,ORI_TYP #VAR,CIRC_TYP #BASE,JERK_FAC 50.0}
DECL FDAT FP550={TOOL_NO 1,BASE_NO 2,IPO_FRAME #BASE,POINT2[] " ",TQ_STATE FALSE}
DECL E6POS XP550={X 598.50634,Y -380.16812,Z 914.54447,A -90,B 0,C 180,S 2,T 35,E1 0,E2 0,E3 0,E4 0,E5 0,E6 0}
; DECL LDAT LCPDATP67={VEL 1,ACC 100,APO_DIST 100,APO_FAC 50.0,ORI_TYP #VAR,CIRC_TYP #BASE,JERK_FAC 50.0}
DECL FDAT FP551={TOOL_NO 1,BASE_NO 2,IPO_FRAME #BASE,POINT2[] " ",TQ_STATE FALSE}
DECL E6POS XP551={X 598.51708,Y -280.17395,Z 814.55076,A -90,B 0,C 180,S 2,T 35,E1 0,E2 0,E3 0,E4 0,E5 0,E6 0}
; DECL PDAT PPDATP35={VEL 100,ACC 100,APO_DIST 100,APO_MODE #CDIS,GEAR_JERK 100.000,EXAX_IGN 0}
DECL FDAT FP552={TOOL_NO 1,BASE_NO 2,IPO_FRAME #BASE,POINT2[] " ",TQ_STATE FALSE}
DECL E6POS XP552={X 598.50603,Y -685.16854,Z 1014.5435,A -90,B 0,C 180,S 2,T 35,E1 0,E2 0,E3 0,E4 0,E5 0,E6 0}
; DECL LDAT LCPDATP68={VEL 1,ACC 100,APO_DIST 100,APO_FAC 50.0,ORI_TYP #VAR,CIRC_TYP #BASE,JERK_FAC 50.0}
DECL FDAT FP553={TOOL_NO 1,BASE_NO 2,IPO_FRAME #BASE,POINT2[] " ",TQ_STATE FALSE}
DECL E6POS XP553={X 598.50693,Y -685.16833,Z 914.54355,A -90,B 0,C 180,S 2,T 35,E1 0,E2 0,E3 0,E4 0,E5 0,E6 0}
; DECL LDAT LCPDATP69={VEL 1,ACC 100,APO_DIST 100,APO_FAC 50.0,ORI_TYP #VAR,CIRC_TYP #BASE,JERK_FAC 50.0}
DECL FDAT FP554={TOOL_NO 1,BASE_NO 2,IPO_FRAME #BASE,POINT2[] " ",TQ_STATE FALSE}
DECL E6POS XP554={X 598.50625,Y -585.16855,Z 814.54416,A -90,B 0,C 180,S 2,T 35,E1 0,E2 0,E3 0,E4 0,E5 0,E6 0}
; ENDDAT for Mtrz_P2_24a28All
; Data for Mtrz_P2_16CoffeCrisp
; DECL PDAT PPDATP51={VEL 100,ACC 100,APO_DIST 100,APO_MODE #CDIS,GEAR_JERK 100.000,EXAX_IGN 0}
DECL FDAT FP564={TOOL_NO 1,BASE_NO 2,IPO_FRAME #BASE,POINT2[] " ",TQ_STATE FALSE}
DECL E6POS XP564={X 1200.44039,Y -690.13163,Z 1019.00134,A -180,B 0,C 180,S 2,T 35,E1 0,E2 0,E3 0,E4 0,E5 0,E6 0}
; DECL LDAT LCPDATP102={VEL 1,ACC 100,APO_DIST 100,APO_FAC 50.0,ORI_TYP #VAR,CIRC_TYP #BASE,JERK_FAC 50.0}
DECL FDAT FP565={TOOL_NO 1,BASE_NO 2,IPO_FRAME #BASE,POINT2[] " ",TQ_STATE FALSE}
DECL E6POS XP565={X 1200.43966,Y -690.13163,Z 892.60201,A -180,B 0,C -180,S 2,T 35,E1 0,E2 0,E3 0,E4 0,E5 0,E6 0}
; DECL LDAT LCPDATP103={VEL 1,ACC 100,APO_DIST 100,APO_FAC 50.0,ORI_TYP #VAR,CIRC_TYP #BASE,JERK_FAC 50.0}
DECL FDAT FP566={TOOL_NO 1,BASE_NO 2,IPO_FRAME #BASE,POINT2[] " ",TQ_STATE FALSE}
DECL E6POS XP566={X 1262.09632,Y -600.00695,Z 814.59915,A 180,B 0,C -180,S 2,T 35,E1 0,E2 0,E3 0,E4 0,E5 0,E6 0}
; DECL PDAT PPDATP52={VEL 100,ACC 100,APO_DIST 100,APO_MODE #CDIS,GEAR_JERK 100.000,EXAX_IGN 0}
DECL FDAT FP567={TOOL_NO 1,BASE_NO 2,IPO_FRAME #BASE,POINT2[] " ",TQ_STATE FALSE}
DECL E6POS XP567={X 799.43993,Y -690.13163,Z 1019.0018,A -180,B 0,C 180,S 2,T 35,E1 0,E2 0,E3 0,E4 0,E5 0,E6 0}
; DECL LDAT LCPDATP104={VEL 1,ACC 100,APO_DIST 100,APO_FAC 50.0,ORI_TYP #VAR,CIRC_TYP #BASE,JERK_FAC 50.0}
DECL FDAT FP568={TOOL_NO 1,BASE_NO 2,IPO_FRAME #BASE,POINT2[] " ",TQ_STATE FALSE}
DECL E6POS XP568={X 799.43989,Y -690.13163,Z 892.60174,A -180,B 0,C -180,S 2,T 35,E1 0,E2 0,E3 0,E4 0,E5 0,E6 0}
; DECL LDAT LCPDATP105={VEL 1,ACC 100,APO_DIST 100,APO_FAC 50.0,ORI_TYP #VAR,CIRC_TYP #BASE,JERK_FAC 50.0}
DECL FDAT FP569={TOOL_NO 1,BASE_NO 2,IPO_FRAME #BASE,POINT2[] " ",TQ_STATE FALSE}
DECL E6POS XP569={X 861.09619,Y -600.00679,Z 814.59921,A 180,B 0,C -180,S 2,T 35,E1 0,E2 0,E3 0,E4 0,E5 0,E6 0}
; DECL PDAT PPDATP53={VEL 100,ACC 100,APO_DIST 100,APO_MODE #CDIS,GEAR_JERK 100.000,EXAX_IGN 0}
DECL FDAT FP570={TOOL_NO 1,BASE_NO 2,IPO_FRAME #BASE,POINT2[] " ",TQ_STATE FALSE}
DECL E6POS XP570={X 398.43905,Y -690.13163,Z 1019.00133,A -180,B 0,C -180,S 2,T 35,E1 0,E2 0,E3 0,E4 0,E5 0,E6 0}
; DECL LDAT LCPDATP106={VEL 1,ACC 100,APO_DIST 100,APO_FAC 50.0,ORI_TYP #VAR,CIRC_TYP #BASE,JERK_FAC 50.0}
DECL FDAT FP571={TOOL_NO 1,BASE_NO 2,IPO_FRAME #BASE,POINT2[] " ",TQ_STATE FALSE}
DECL E6POS XP571={X 398.4393,Y -690.13163,Z 892.60169,A 180,B 0,C -180,S 2,T 35,E1 0,E2 0,E3 0,E4 0,E5 0,E6 0}
; DECL LDAT LCPDATP107={VEL 1,ACC 100,APO_DIST 100,APO_FAC 50.0,ORI_TYP #VAR,CIRC_TYP #BASE,JERK_FAC 50.0}
DECL FDAT FP572={TOOL_NO 1,BASE_NO 2,IPO_FRAME #BASE,POINT2[] " ",TQ_STATE FALSE}
DECL E6POS XP572={X 460.09604,Y -600.00686,Z 814.59882,A -180,B 0,C -180,S 2,T 35,E1 0,E2 0,E3 0,E4 0,E5 0,E6 0}
; DECL PDAT PPDATP54={VEL 100,ACC 100,APO_DIST 100,APO_MODE #CDIS,GEAR_JERK 100.000,EXAX_IGN 0}
DECL FDAT FP573={TOOL_NO 1,BASE_NO 2,IPO_FRAME #BASE,POINT2[] " ",TQ_STATE FALSE}
DECL E6POS XP573={X 603.07783,Y -590.51697,Z 1019.00114,A -90,B 0,C 180,S 2,T 35,E1 0,E2 0,E3 0,E4 0,E5 0,E6 0}
; DECL LDAT LCPDATP108={VEL 1,ACC 100,APO_DIST 100,APO_FAC 50.0,ORI_TYP #VAR,CIRC_TYP #BASE,JERK_FAC 50.0}
DECL FDAT FP574={TOOL_NO 1,BASE_NO 2,IPO_FRAME #BASE,POINT2[] " ",TQ_STATE FALSE}
DECL E6POS XP574={X 603.0778,Y -590.51676,Z 969.00176,A -90,B 0,C 180,S 2,T 35,E1 0,E2 0,E3 0,E4 0,E5 0,E6 0}
; DECL LDAT LCPDATP109={VEL 1,ACC 100,APO_DIST 100,APO_FAC 50.0,ORI_TYP #VAR,CIRC_TYP #BASE,JERK_FAC 50.0}
DECL FDAT FP575={TOOL_NO 1,BASE_NO 2,IPO_FRAME #BASE,POINT2[] " ",TQ_STATE FALSE}
DECL E6POS XP575={X 603.07772,Y -540.51695,Z 814.5989,A -90,B 0,C 180,S 2,T 35,E1 0,E2 0,E3 0,E4 0,E5 0,E6 0}
; DECL PDAT PPDATP55={VEL 100,ACC 100,APO_DIST 100,APO_MODE #CDIS,GEAR_JERK 100.000,EXAX_IGN 0}
DECL FDAT FP576={TOOL_NO 1,BASE_NO 2,IPO_FRAME #BASE,POINT2[] " ",TQ_STATE FALSE}
DECL E6POS XP576={X 603.08186,Y 9.46734,Z 1084.57819,A -90,B 0,C 180,S 2,T 35,E1 0,E2 0,E3 0,E4 0,E5 0,E6 0}
; DECL LDAT LCPDATP110={VEL 1,ACC 100,APO_DIST 100,APO_FAC 50.0,ORI_TYP #VAR,CIRC_TYP #BASE,JERK_FAC 50.0}
DECL FDAT FP577={TOOL_NO 1,BASE_NO 2,IPO_FRAME #BASE,POINT2[] " ",TQ_STATE FALSE}
DECL E6POS XP577={X 603.08184,Y 9.4675,Z 1064.57625,A -90,B 0,C 180,S 2,T 35,E1 0,E2 0,E3 0,E4 0,E5 0,E6 0}
; DECL LDAT LCPDATP111={VEL 1,ACC 100,APO_DIST 100,APO_FAC 50.0,ORI_TYP #VAR,CIRC_TYP #BASE,JERK_FAC 50.0}
DECL FDAT FP578={TOOL_NO 1,BASE_NO 2,IPO_FRAME #BASE,POINT2[] " ",TQ_STATE FALSE}
DECL E6POS XP578={X 603.08152,Y 59.46749,Z 964.58333,A -90,B 0,C 180,S 2,T 35,E1 0,E2 0,E3 0,E4 0,E5 0,E6 0}
; DECL PDAT PPDATP59={VEL 100,ACC 100,APO_DIST 100,APO_MODE #CDIS,GEAR_JERK 100.000,EXAX_IGN 0}
DECL FDAT FP579={TOOL_NO 1,BASE_NO 2,IPO_FRAME #BASE,POINT2[] " ",TQ_STATE FALSE}
DECL E6POS XP579={X 1212.09936,Y -1051.03809,Z 1164.57839,A -180,B 0,C 180,S 2,T 35,E1 0,E2 0,E3 0,E4 0,E5 0,E6 0}
; DECL LDAT LCPDATP112={VEL 1,ACC 100,APO_DIST 100,APO_FAC 50.0,ORI_TYP #VAR,CIRC_TYP #BASE,JERK_FAC 50.0}
DECL FDAT FP580={TOOL_NO 1,BASE_NO 2,IPO_FRAME #BASE,POINT2[] " ",TQ_STATE FALSE}
DECL E6POS XP580={X 1212.09934,Y -1051.03809,Z 1064.59787,A -180,B 0,C 180,S 2,T 35,E1 0,E2 0,E3 0,E4 0,E5 0,E6 0}
; DECL LDAT LCPDATP113={VEL 1,ACC 100,APO_DIST 100,APO_FAC 50.0,ORI_TYP #VAR,CIRC_TYP #BASE,JERK_FAC 50.0}
DECL FDAT FP581={TOOL_NO 1,BASE_NO 2,IPO_FRAME #BASE,POINT2[] " ",TQ_STATE FALSE}
DECL E6POS XP581={X 1262.09971,Y -1001.04492,Z 964.59722,A 180,B 0,C 180,S 2,T 35,E1 0,E2 0,E3 0,E4 0,E5 0,E6 0}
; DECL PDAT PPDATP57={VEL 100,ACC 100,APO_DIST 100,APO_MODE #CDIS,GEAR_JERK 100.000,EXAX_IGN 0}
DECL FDAT FP582={TOOL_NO 1,BASE_NO 2,IPO_FRAME #BASE,POINT2[] " ",TQ_STATE FALSE}
DECL E6POS XP582={X 811.09468,Y -1051.03809,Z 1164.57844,A -180,B 0,C -180,S 2,T 35,E1 0,E2 0,E3 0,E4 0,E5 0,E6 0}
; DECL LDAT LCPDATP114={VEL 1,ACC 100,APO_DIST 100,APO_FAC 50.0,ORI_TYP #VAR,CIRC_TYP #BASE,JERK_FAC 50.0}
DECL FDAT FP583={TOOL_NO 1,BASE_NO 2,IPO_FRAME #BASE,POINT2[] " ",TQ_STATE FALSE}
DECL E6POS XP583={X 811.09431,Y -1051.03809,Z 1064.59749,A -180,B 0,C 180,S 2,T 35,E1 0,E2 0,E3 0,E4 0,E5 0,E6 0}
; DECL LDAT LCPDATP115={VEL 1,ACC 100,APO_DIST 100,APO_FAC 50.0,ORI_TYP #VAR,CIRC_TYP #BASE,JERK_FAC 50.0}
DECL FDAT FP584={TOOL_NO 1,BASE_NO 2,IPO_FRAME #BASE,POINT2[] " ",TQ_STATE FALSE}
DECL E6POS XP584={X 861.09415,Y -1001.03503,Z 964.60474,A 180,B 0,C -180,S 2,T 35,E1 0,E2 0,E3 0,E4 0,E5 0,E6 0}
; DECL PDAT PPDATP58={VEL 100,ACC 100,APO_DIST 100,APO_MODE #CDIS,GEAR_JERK 100.000,EXAX_IGN 0}
DECL FDAT FP585={TOOL_NO 1,BASE_NO 2,IPO_FRAME #BASE,POINT2[] " ",TQ_STATE FALSE}
DECL E6POS XP585={X 410.09422,Y -1051.03809,Z 1164.59982,A -180,B 0,C -180,S 2,T 35,E1 0,E2 0,E3 0,E4 0,E5 0,E6 0}
; DECL LDAT LCPDATP116={VEL 1,ACC 100,APO_DIST 100,APO_FAC 50.0,ORI_TYP #VAR,CIRC_TYP #BASE,JERK_FAC 50.0}
DECL FDAT FP586={TOOL_NO 1,BASE_NO 2,IPO_FRAME #BASE,POINT2[] " ",TQ_STATE FALSE}
DECL E6POS XP586={X 410.09432,Y -1051.03809,Z 1064.60018,A 180,B 0,C -180,S 2,T 35,E1 0,E2 0,E3 0,E4 0,E5 0,E6 0}
; DECL LDAT LCPDATP117={VEL 1,ACC 100,APO_DIST 100,APO_FAC 50.0,ORI_TYP #VAR,CIRC_TYP #BASE,JERK_FAC 50.0}
DECL FDAT FP587={TOOL_NO 1,BASE_NO 2,IPO_FRAME #BASE,POINT2[] " ",TQ_STATE FALSE}
DECL E6POS XP587={X 460.09451,Y -1001.03794,Z 964.60836,A -180,B 0,C 180,S 2,T 35,E1 0,E2 0,E3 0,E4 0,E5 0,E6 0}
; ENDDAT for Mtrz_P2_16CoffeCrisp
; Data for Mtrz_P2_37BarPacking
; DECL PDAT PPDATP19={VEL 100,ACC 100,APO_DIST 100,APO_MODE #CDIS,GEAR_JERK 100.000,EXAX_IGN 0}
DECL FDAT FP588={TOOL_NO 1,BASE_NO 2,IPO_FRAME #BASE,POINT2[] " ",TQ_STATE FALSE}
DECL E6POS XP588={X 557.61101,Y -111.61638,Z 1263.48407,A -90,B 0,C 180,S 2,T 35,E1 0,E2 0,E3 0,E4 0,E5 0,E6 0}
; DECL LDAT LCPDATP36={VEL 1,ACC 100,APO_DIST 100,APO_FAC 50.0,ORI_TYP #VAR,CIRC_TYP #BASE,JERK_FAC 50.0}
DECL FDAT FP589={TOOL_NO 1,BASE_NO 2,IPO_FRAME #BASE,POINT2[] " ",TQ_STATE FALSE}
DECL E6POS XP589={X 557.61102,Y -111.61645,Z 1063.48526,A -90,B 0,C 180,S 2,T 35,E1 0,E2 0,E3 0,E4 0,E5 0,E6 0}
; DECL LDAT LCPDATP37={VEL 1,ACC 100,APO_DIST 100,APO_FAC 50.0,ORI_TYP #VAR,CIRC_TYP #BASE,JERK_FAC 50.0}
DECL FDAT FP590={TOOL_NO 1,BASE_NO 2,IPO_FRAME #BASE,POINT2[] " ",TQ_STATE FALSE}
DECL E6POS XP590={X 557.6118,Y -11.61642,Z 863.48454,A -90,B 0,C 180,S 2,T 35,E1 0,E2 0,E3 0,E4 0,E5 0,E6 0}
; DECL PDAT PPDATP20={VEL 100,ACC 100,APO_DIST 100,APO_MODE #CDIS,GEAR_JERK 100.000,EXAX_IGN 0}
DECL FDAT FP591={TOOL_NO 1,BASE_NO 2,IPO_FRAME #BASE,POINT2[] " ",TQ_STATE FALSE}
DECL E6POS XP591={X 557.61163,Y -607.61597,Z 1263.48456,A -90,B 0,C 180,S 2,T 35,E1 0,E2 0,E3 0,E4 0,E5 0,E6 0}
; DECL LDAT LCPDATP38={VEL 1,ACC 100,APO_DIST 100,APO_FAC 50.0,ORI_TYP #VAR,CIRC_TYP #BASE,JERK_FAC 50.0}
DECL FDAT FP592={TOOL_NO 1,BASE_NO 2,IPO_FRAME #BASE,POINT2[] " ",TQ_STATE FALSE}
DECL E6POS XP592={X 557.61169,Y -607.61647,Z 1063.48493,A -90,B 0,C 180,S 2,T 35,E1 0,E2 0,E3 0,E4 0,E5 0,E6 0}
; DECL LDAT LCPDATP39={VEL 1,ACC 100,APO_DIST 100,APO_FAC 50.0,ORI_TYP #VAR,CIRC_TYP #BASE,JERK_FAC 50.0}
DECL FDAT FP593={TOOL_NO 1,BASE_NO 2,IPO_FRAME #BASE,POINT2[] " ",TQ_STATE FALSE}
DECL E6POS XP593={X 557.61131,Y -507.61657,Z 863.4846,A -90,B 0,C 180,S 2,T 35,E1 0,E2 0,E3 0,E4 0,E5 0,E6 0}
; ENDDAT for Mtrz_P2_37BarPacking
; Data for Pick_E_2_P_2
; DECL PDAT PPDATP1={VEL 100,ACC 100,APO_DIST 100,APO_MODE #CDIS,GEAR_JERK 100.000,EXAX_IGN 0}
DECL FDAT FP600={TOOL_NO 1,BASE_NO 4,IPO_FRAME #BASE,POINT2[] " ",TQ_STATE FALSE}
DECL E6POS XP600={X 542.90832,Y 2.83153,Z 2105.80075,A -90,B 0,C -180,S 2,T 3,E1 0,E2 0,E3 0,E4 0,E5 0,E6 0}
; DECL LDAT LCPDATP2={VEL 1,ACC 100,APO_DIST 100,APO_FAC 50.0,ORI_TYP #VAR,CIRC_TYP #BASE,JERK_FAC 50.0}
DECL FDAT FP601={TOOL_NO 1,BASE_NO 4,IPO_FRAME #BASE,POINT2[] " ",TQ_STATE FALSE}
DECL E6POS XP601={X 542.90832,Y 2.83193,Z 1391.79999,A -90,B 0,C -180,S 2,T 3,E1 0,E2 0,E3 0,E4 0,E5 0,E6 0}
; DECL LDAT LCPDATP1={VEL 1,ACC 100,APO_DIST 100,APO_FAC 50.0,ORI_TYP #VAR,CIRC_TYP #BASE,JERK_FAC 50.0}
DECL FDAT FPick_E_2_P_2={TOOL_NO 1,BASE_NO 4,IPO_FRAME #BASE,POINT2[] " ",TQ_STATE FALSE}
DECL E6POS XPick_E_2_P_2={X 542.90832,Y -19.40194,Z 1391.79999,A -90,B 0,C 180,S 2,T 3,E1 0,E2 0,E3 0,E4 0,E5 0,E6 0}
; DECL LDAT LCPDATP3={VEL 1,ACC 100,APO_DIST 100,APO_FAC 50.0,ORI_TYP #VAR,CIRC_TYP #BASE,JERK_FAC 50.0}
DECL FDAT FP603={TOOL_NO 1,BASE_NO 4,IPO_FRAME #BASE,POINT2[] " ",TQ_STATE FALSE}
DECL E6POS XP603={X 542.90832,Y -19.40201,Z 2105.79999,A -90,B 0,C -180,S 2,T 3,E1 0,E2 0,E3 0,E4 0,E5 0,E6 0}
; ENDDAT for Pick_E_2_P_2
; Data for Mtrz_P2_36BarPacking
; DECL PDAT PPDATP21={VEL 100,ACC 100,APO_DIST 100,APO_MODE #CDIS,GEAR_JERK 100.000,EXAX_IGN 0}
DECL FDAT FP602={TOOL_NO 1,BASE_NO 2,IPO_FRAME #BASE,POINT2[] " ",TQ_STATE FALSE}
DECL E6POS XP602={X 562.60865,Y -356.53512,Z 1263.45992,A -90,B 0,C 180,S 2,T 35,E1 0,E2 0,E3 0,E4 0,E5 0,E6 0}
; DECL LDAT LCPDATP40={VEL 1,ACC 100,APO_DIST 100,APO_FAC 50.0,ORI_TYP #VAR,CIRC_TYP #BASE,JERK_FAC 50.0}
DECL FDAT FP604={TOOL_NO 1,BASE_NO 2,IPO_FRAME #BASE,POINT2[] " ",TQ_STATE FALSE}
DECL E6POS XP604={X 562.6086,Y -356.53471,Z 1063.46026,A -90,B 0,C 180,S 2,T 35,E1 0,E2 0,E3 0,E4 0,E5 0,E6 0}
; DECL LDAT LCPDATP41={VEL 1,ACC 100,APO_DIST 100,APO_FAC 50.0,ORI_TYP #VAR,CIRC_TYP #BASE,JERK_FAC 50.0}
DECL FDAT FP605={TOOL_NO 1,BASE_NO 2,IPO_FRAME #BASE,POINT2[] " ",TQ_STATE FALSE}
DECL E6POS XP605={X 562.60916,Y -256.53557,Z 863.45968,A -90,B 0,C 180,S 2,T 35,E1 0,E2 0,E3 0,E4 0,E5 0,E6 0}
; ENDDAT for Mtrz_P2_36BarPacking
; Data for Mtrz_P2_22KitKat
; DECL PDAT PPDATP36={VEL 100,ACC 100,APO_DIST 100,APO_MODE #CDIS,GEAR_JERK 100.000,EXAX_IGN 0}
DECL FDAT FP606={TOOL_NO 1,BASE_NO 2,IPO_FRAME #BASE,POINT2[] " ",TQ_STATE FALSE}
DECL E6POS XP606={X 1066.23936,Y -555.93148,Z 1141.50167,A -180,B 0,C -180,S 2,T 35,E1 0,E2 0,E3 0,E4 0,E5 0,E6 0}
; DECL LDAT LCPDATP70={VEL 1,ACC 100,APO_DIST 100,APO_FAC 50.0,ORI_TYP #VAR,CIRC_TYP #BASE,JERK_FAC 50.0}
DECL FDAT FP607={TOOL_NO 1,BASE_NO 2,IPO_FRAME #BASE,POINT2[] " ",TQ_STATE FALSE}
DECL E6POS XP607={X 1066.23956,Y -555.93156,Z 941.50237,A -180,B 0,C -180,S 2,T 35,E1 0,E2 0,E3 0,E4 0,E5 0,E6 0}
; DECL LDAT LCPDATP71={VEL 1,ACC 100,APO_DIST 100,APO_FAC 50.0,ORI_TYP #VAR,CIRC_TYP #BASE,JERK_FAC 50.0}
DECL FDAT FP608={TOOL_NO 1,BASE_NO 2,IPO_FRAME #BASE,POINT2[] " ",TQ_STATE FALSE}
DECL E6POS XP608={X 1166.24033,Y -555.93147,Z 841.5026,A 180,B 0,C -180,S 2,T 35,E1 0,E2 0,E3 0,E4 0,E5 0,E6 0}
; DECL PDAT PPDATP37={VEL 100,ACC 100,APO_DIST 100,APO_MODE #CDIS,GEAR_JERK 100.000,EXAX_IGN 0}
DECL FDAT FP609={TOOL_NO 1,BASE_NO 2,IPO_FRAME #BASE,POINT2[] " ",TQ_STATE FALSE}
DECL E6POS XP609={X 672.23914,Y -555.93167,Z 1141.50271,A -180,B 0,C -180,S 2,T 35,E1 0,E2 0,E3 0,E4 0,E5 0,E6 0}
; DECL LDAT LCPDATP72={VEL 1,ACC 100,APO_DIST 100,APO_FAC 50.0,ORI_TYP #VAR,CIRC_TYP #BASE,JERK_FAC 50.0}
DECL FDAT FP610={TOOL_NO 1,BASE_NO 2,IPO_FRAME #BASE,POINT2[] " ",TQ_STATE FALSE}
DECL E6POS XP610={X 672.23959,Y -555.93151,Z 941.50181,A 180,B 0,C -180,S 2,T 35,E1 0,E2 0,E3 0,E4 0,E5 0,E6 0}
; DECL LDAT LCPDATP73={VEL 1,ACC 100,APO_DIST 100,APO_FAC 50.0,ORI_TYP #VAR,CIRC_TYP #BASE,JERK_FAC 50.0}
DECL FDAT FP611={TOOL_NO 1,BASE_NO 2,IPO_FRAME #BASE,POINT2[] " ",TQ_STATE FALSE}
DECL E6POS XP611={X 772.24013,Y -555.93149,Z 841.50209,A -180,B 0,C 180,S 2,T 35,E1 0,E2 0,E3 0,E4 0,E5 0,E6 0}
; DECL PDAT PPDATP38={VEL 100,ACC 100,APO_DIST 100,APO_MODE #CDIS,GEAR_JERK 100.000,EXAX_IGN 0}
DECL FDAT FP612={TOOL_NO 1,BASE_NO 2,IPO_FRAME #BASE,POINT2[] " ",TQ_STATE FALSE}
DECL E6POS XP612={X 328.23921,Y -555.93135,Z 1141.50226,A -180,B 0,C -180,S 2,T 35,E1 0,E2 0,E3 0,E4 0,E5 0,E6 0}
; DECL LDAT LCPDATP74={VEL 1,ACC 100,APO_DIST 100,APO_FAC 50.0,ORI_TYP #VAR,CIRC_TYP #BASE,JERK_FAC 50.0}
DECL FDAT FP613={TOOL_NO 1,BASE_NO 2,IPO_FRAME #BASE,POINT2[] " ",TQ_STATE FALSE}
DECL E6POS XP613={X 328.23968,Y -555.9315,Z 941.50171,A -180,B 0,C -180,S 2,T 35,E1 0,E2 0,E3 0,E4 0,E5 0,E6 0}
; DECL LDAT LCPDATP75={VEL 1,ACC 100,APO_DIST 100,APO_FAC 50.0,ORI_TYP #VAR,CIRC_TYP #BASE,JERK_FAC 50.0}
DECL FDAT FP614={TOOL_NO 1,BASE_NO 2,IPO_FRAME #BASE,POINT2[] " ",TQ_STATE FALSE}
DECL E6POS XP614={X 378.23966,Y -555.93116,Z 841.50213,A -180,B 0,C -180,S 2,T 35,E1 0,E2 0,E3 0,E4 0,E5 0,E6 0}
; DECL PDAT PPDATP44={VEL 100,ACC 100,APO_DIST 100,APO_MODE #CDIS,GEAR_JERK 100.000,EXAX_IGN 0}
DECL FDAT FP615={TOOL_NO 1,BASE_NO 2,IPO_FRAME #BASE,POINT2[] " ",TQ_STATE FALSE}
DECL E6POS XP615={X 563.18108,Y -658.59718,Z 1167.90221,A -90,B 0,C 180,S 2,T 35,E1 0,E2 0,E3 0,E4 0,E5 0,E6 0}
; DECL LDAT LCPDATP77={VEL 1,ACC 100,APO_DIST 100,APO_FAC 50.0,ORI_TYP #VAR,CIRC_TYP #BASE,JERK_FAC 50.0}
DECL FDAT FP616={TOOL_NO 1,BASE_NO 2,IPO_FRAME #BASE,POINT2[] " ",TQ_STATE FALSE}
DECL E6POS XP616={X 563.1811,Y -658.59734,Z 1041.51047,A -90,B 0,C 180,S 2,T 35,E1 0,E2 0,E3 0,E4 0,E5 0,E6 0}
; DECL LDAT LCPDATP86={VEL 1,ACC 100,APO_DIST 100,APO_FAC 50.0,ORI_TYP #VAR,CIRC_TYP #BASE,JERK_FAC 50.0}
DECL FDAT FP617={TOOL_NO 1,BASE_NO 2,IPO_FRAME #BASE,POINT2[] " ",TQ_STATE FALSE}
DECL E6POS XP617={X 563.1807,Y -608.59735,Z 841.51045,A -90,B 0,C 180,S 2,T 35,E1 0,E2 0,E3 0,E4 0,E5 0,E6 0}
; DECL PDAT PPDATP40={VEL 100,ACC 100,APO_DIST 100,APO_MODE #CDIS,GEAR_JERK 100.000,EXAX_IGN 0}
DECL FDAT FP618={TOOL_NO 1,BASE_NO 2,IPO_FRAME #BASE,POINT2[] " ",TQ_STATE FALSE}
DECL E6POS XP618={X 563.18297,Y -180.42867,Z 1300.9019,A -90,B 0,C 180,S 2,T 35,E1 0,E2 0,E3 0,E4 0,E5 0,E6 0}
; DECL LDAT LCPDATP78={VEL 1,ACC 100,APO_DIST 100,APO_FAC 50.0,ORI_TYP #VAR,CIRC_TYP #BASE,JERK_FAC 50.0}
DECL FDAT FP619={TOOL_NO 1,BASE_NO 2,IPO_FRAME #BASE,POINT2[] " ",TQ_STATE FALSE}
DECL E6POS XP619={X 563.18303,Y -180.42922,Z 1200.90196,A -90,B 0,C 180,S 2,T 35,E1 0,E2 0,E3 0,E4 0,E5 0,E6 0}
; DECL LDAT LCPDATP79={VEL 1,ACC 100,APO_DIST 100,APO_FAC 50.0,ORI_TYP #VAR,CIRC_TYP #BASE,JERK_FAC 50.0}
DECL FDAT FP620={TOOL_NO 1,BASE_NO 2,IPO_FRAME #BASE,POINT2[] " ",TQ_STATE FALSE}
DECL E6POS XP620={X 563.18269,Y -26.61185,Z 1074.50219,A -90,B 0,C 180,S 2,T 35,E1 0,E2 0,E3 0,E4 0,E5 0,E6 0}
; DECL PDAT PPDATP41={VEL 100,ACC 100,APO_DIST 100,APO_MODE #CDIS,GEAR_JERK 100.000,EXAX_IGN 0}
DECL FDAT FP621={TOOL_NO 1,BASE_NO 2,IPO_FRAME #BASE,POINT2[] " ",TQ_STATE FALSE}
DECL E6POS XP621={X 1116.24422,Y -981.19257,Z 1350.90082,A -180,B 0,C -180,S 2,T 35,E1 0,E2 0,E3 0,E4 0,E5 0,E6 0}
; DECL LDAT LCPDATP80={VEL 1,ACC 100,APO_DIST 100,APO_FAC 50.0,ORI_TYP #VAR,CIRC_TYP #BASE,JERK_FAC 50.0}
DECL FDAT FP622={TOOL_NO 1,BASE_NO 2,IPO_FRAME #BASE,POINT2[] " ",TQ_STATE FALSE}
DECL E6POS XP622={X 1116.24389,Y -981.19257,Z 1200.90198,A 180,B 0,C 180,S 2,T 35,E1 0,E2 0,E3 0,E4 0,E5 0,E6 0}
; DECL LDAT LCPDATP81={VEL 1,ACC 100,APO_DIST 100,APO_FAC 50.0,ORI_TYP #VAR,CIRC_TYP #BASE,JERK_FAC 50.0}
DECL FDAT FP623={TOOL_NO 1,BASE_NO 2,IPO_FRAME #BASE,POINT2[] " ",TQ_STATE FALSE}
DECL E6POS XP623={X 1166.24386,Y -931.19259,Z 1074.50233,A 180,B 0,C 180,S 2,T 35,E1 0,E2 0,E3 0,E4 0,E5 0,E6 0}
; DECL PDAT PPDATP42={VEL 100,ACC 100,APO_DIST 100,APO_MODE #CDIS,GEAR_JERK 100.000,EXAX_IGN 0}
DECL FDAT FP624={TOOL_NO 1,BASE_NO 2,IPO_FRAME #BASE,POINT2[] " ",TQ_STATE FALSE}
DECL E6POS XP624={X 721.67962,Y -981.19257,Z 1350.90102,A -180,B 0,C 180,S 2,T 35,E1 0,E2 0,E3 0,E4 0,E5 0,E6 0}
; DECL LDAT LCPDATP82={VEL 1,ACC 100,APO_DIST 100,APO_FAC 50.0,ORI_TYP #VAR,CIRC_TYP #BASE,JERK_FAC 50.0}
DECL FDAT FP625={TOOL_NO 1,BASE_NO 2,IPO_FRAME #BASE,POINT2[] " ",TQ_STATE FALSE}
DECL E6POS XP625={X 721.6796,Y -981.19257,Z 1200.90226,A 180,B 0,C 180,S 2,T 35,E1 0,E2 0,E3 0,E4 0,E5 0,E6 0}
; DECL LDAT LCPDATP84={VEL 1,ACC 100,APO_DIST 100,APO_FAC 50.0,ORI_TYP #VAR,CIRC_TYP #BASE,JERK_FAC 50.0}
DECL FDAT FP626={TOOL_NO 1,BASE_NO 2,IPO_FRAME #BASE,POINT2[] " ",TQ_STATE FALSE}
DECL E6POS XP626={X 771.67974,Y -931.19212,Z 1074.49963,A 180,B 0,C -180,S 2,T 35,E1 0,E2 0,E3 0,E4 0,E5 0,E6 0}
; DECL PDAT PPDATP43={VEL 100,ACC 100,APO_DIST 100,APO_MODE #CDIS,GEAR_JERK 100.000,EXAX_IGN 0}
DECL FDAT FP627={TOOL_NO 1,BASE_NO 2,IPO_FRAME #BASE,POINT2[] " ",TQ_STATE FALSE}
DECL E6POS XP627={X 325.24329,Y -981.19257,Z 1350.90233,A -180,B 0,C -180,S 2,T 35,E1 0,E2 0,E3 0,E4 0,E5 0,E6 0}
; DECL LDAT LCPDATP83={VEL 1,ACC 100,APO_DIST 100,APO_FAC 50.0,ORI_TYP #VAR,CIRC_TYP #BASE,JERK_FAC 50.0}
DECL FDAT FP628={TOOL_NO 1,BASE_NO 2,IPO_FRAME #BASE,POINT2[] " ",TQ_STATE FALSE}
DECL E6POS XP628={X 325.24344,Y -981.19257,Z 1200.90192,A 180,B 0,C 180,S 2,T 35,E1 0,E2 0,E3 0,E4 0,E5 0,E6 0}
; DECL LDAT LCPDATP85={VEL 1,ACC 100,APO_DIST 100,APO_FAC 50.0,ORI_TYP #VAR,CIRC_TYP #BASE,JERK_FAC 50.0}
DECL FDAT FP629={TOOL_NO 1,BASE_NO 2,IPO_FRAME #BASE,POINT2[] " ",TQ_STATE FALSE}
DECL E6POS XP629={X 375.24327,Y -931.19248,Z 1074.50198,A 180,B 0,C 180,S 2,T 35,E1 0,E2 0,E3 0,E4 0,E5 0,E6 0}
; ENDDAT for Mtrz_P2_22KitKat
; Data for Mtrz_P2_35BarPacking
; DECL PDAT PPDATP47={VEL 100,ACC 100,APO_DIST 100,APO_MODE #CDIS,GEAR_JERK 100.000,EXAX_IGN 0}
DECL FDAT FP630={TOOL_NO 1,BASE_NO 2,IPO_FRAME #BASE,POINT2[] " ",TQ_STATE FALSE}
DECL E6POS XP630={X 1128.19567,Y -552.20825,Z 1215.66303,A -180,B 0,C 180,S 2,T 35,E1 0,E2 0,E3 0,E4 0,E5 0,E6 0}
; DECL LDAT LCPDATP92={VEL 1,ACC 100,APO_DIST 100,APO_FAC 50.0,ORI_TYP #VAR,CIRC_TYP #BASE,JERK_FAC 50.0}
DECL FDAT FP631={TOOL_NO 1,BASE_NO 2,IPO_FRAME #BASE,POINT2[] " ",TQ_STATE FALSE}
DECL E6POS XP631={X 1128.19623,Y -552.20835,Z 1015.66288,A 180,B 0,C 180,S 2,T 35,E1 0,E2 0,E3 0,E4 0,E5 0,E6 0}
; DECL LDAT LCPDATP93={VEL 1,ACC 100,APO_DIST 100,APO_FAC 50.0,ORI_TYP #VAR,CIRC_TYP #BASE,JERK_FAC 50.0}
DECL FDAT FP632={TOOL_NO 1,BASE_NO 2,IPO_FRAME #BASE,POINT2[] " ",TQ_STATE FALSE}
DECL E6POS XP632={X 1178.19625,Y -552.20835,Z 865.66289,A -180,B 0,C -180,S 2,T 35,E1 0,E2 0,E3 0,E4 0,E5 0,E6 0}
; DECL PDAT PPDATP48={VEL 100,ACC 100,APO_DIST 100,APO_MODE #CDIS,GEAR_JERK 100.000,EXAX_IGN 0}
DECL FDAT FP633={TOOL_NO 1,BASE_NO 2,IPO_FRAME #BASE,POINT2[] " ",TQ_STATE FALSE}
DECL E6POS XP633={X 532.19535,Y -552.20804,Z 1215.66364,A -180,B 0,C -180,S 2,T 35,E1 0,E2 0,E3 0,E4 0,E5 0,E6 0}
; DECL LDAT LCPDATP95={VEL 1,ACC 100,APO_DIST 100,APO_FAC 50.0,ORI_TYP #VAR,CIRC_TYP #BASE,JERK_FAC 50.0}
DECL FDAT FP634={TOOL_NO 1,BASE_NO 2,IPO_FRAME #BASE,POINT2[] " ",TQ_STATE FALSE}
DECL E6POS XP634={X 532.19539,Y -552.20804,Z 1015.66268,A -180,B 0,C -180,S 2,T 35,E1 0,E2 0,E3 0,E4 0,E5 0,E6 0}
; DECL LDAT LCPDATP94={VEL 1,ACC 100,APO_DIST 100,APO_FAC 50.0,ORI_TYP #VAR,CIRC_TYP #BASE,JERK_FAC 50.0}
DECL FDAT FP635={TOOL_NO 1,BASE_NO 2,IPO_FRAME #BASE,POINT2[] " ",TQ_STATE FALSE}
DECL E6POS XP635={X 582.19539,Y -552.20804,Z 865.66281,A -180,B 0,C 180,S 2,T 35,E1 0,E2 0,E3 0,E4 0,E5 0,E6 0}
; DECL PDAT PPDATP49={VEL 100,ACC 100,APO_DIST 100,APO_MODE #CDIS,GEAR_JERK 100.000,EXAX_IGN 0}
DECL FDAT FP636={TOOL_NO 1,BASE_NO 2,IPO_FRAME #BASE,POINT2[] " ",TQ_STATE FALSE}
DECL E6POS XP636={X 569.41677,Y -557.00625,Z 1274.46311,A -90,B 0,C 180,S 2,T 35,E1 0,E2 0,E3 0,E4 0,E5 0,E6 0}
; DECL LDAT LCPDATP96={VEL 1,ACC 100,APO_DIST 100,APO_FAC 50.0,ORI_TYP #VAR,CIRC_TYP #BASE,JERK_FAC 50.0}
DECL FDAT FP637={TOOL_NO 1,BASE_NO 2,IPO_FRAME #BASE,POINT2[] " ",TQ_STATE FALSE}
DECL E6POS XP637={X 569.41678,Y -557.0063,Z 1024.46326,A -90,B 0,C 180,S 2,T 35,E1 0,E2 0,E3 0,E4 0,E5 0,E6 0}
; DECL LDAT LCPDATP97={VEL 1,ACC 100,APO_DIST 100,APO_FAC 50.0,ORI_TYP #VAR,CIRC_TYP #BASE,JERK_FAC 50.0}
DECL FDAT FP638={TOOL_NO 1,BASE_NO 2,IPO_FRAME #BASE,POINT2[] " ",TQ_STATE FALSE}
DECL E6POS XP638={X 569.41676,Y -409.86988,Z 865.6385,A -90,B 0,C 180,S 2,T 35,E1 0,E2 0,E3 0,E4 0,E5 0,E6 0}
; ENDDAT for Mtrz_P2_35BarPacking
; Data for Pick_E_1_P_2_3
; DECL PDAT PPDATP1={VEL 100,ACC 100,APO_DIST 100,APO_MODE #CDIS,GEAR_JERK 100.000,EXAX_IGN 0}
DECL FDAT FP78={TOOL_NO 1,BASE_NO 3,IPO_FRAME #BASE,POINT2[] " ",TQ_STATE FALSE}
DECL E6POS XP78={X 548.60753,Y -2.83256,Z 2105.79953,A 90,B 0,C -180,S 2,T 34,E1 0,E2 0,E3 0,E4 0,E5 0,E6 0}
; DECL LDAT LCPDATP2={VEL 1,ACC 100,APO_DIST 100,APO_FAC 50.0,ORI_TYP #VAR,CIRC_TYP #BASE,JERK_FAC 50.0}
DECL FDAT FP294={TOOL_NO 1,BASE_NO 3,IPO_FRAME #BASE,POINT2[] " ",TQ_STATE FALSE}
DECL E6POS XP294={X 548.60753,Y -2.8321,Z 1392.47867,A 90,B 0,C -180,S 2,T 34,E1 0,E2 0,E3 0,E4 0,E5 0,E6 0}
; DECL LDAT LCPDATP1={VEL 1,ACC 100,APO_DIST 100,APO_FAC 50.0,ORI_TYP #VAR,CIRC_TYP #BASE,JERK_FAC 50.0}
DECL FDAT FPick_E_1_P_2_3={TOOL_NO 1,BASE_NO 3,IPO_FRAME #BASE,POINT2[] " ",TQ_STATE FALSE}
DECL E6POS XPick_E_1_P_2_3={X 548.60753,Y 19.40185,Z 1392.47867,A 90,B 0,C -180,S 2,T 34,E1 0,E2 0,E3 0,E4 0,E5 0,E6 0}
; DECL LDAT LCPDATP3={VEL 1,ACC 100,APO_DIST 100,APO_FAC 50.0,ORI_TYP #VAR,CIRC_TYP #BASE,JERK_FAC 50.0}
DECL FDAT FP295={TOOL_NO 1,BASE_NO 3,IPO_FRAME #BASE,POINT2[] " ",TQ_STATE FALSE}
DECL E6POS XP295={X 548.60753,Y 19.40185,Z 2105.80057,A 90,B 0,C 180,S 2,T 34,E1 0,E2 0,E3 0,E4 0,E5 0,E6 0}
; ENDDAT for Pick_E_1_P_2_3
; Data for Mtrz_P2_32BarPacking
; DECL PDAT PPDATP22={VEL 100,ACC 100,APO_DIST 100,APO_MODE #CDIS,GEAR_JERK 100.000,EXAX_IGN 0}
DECL FDAT FP296={TOOL_NO 1,BASE_NO 2,IPO_FRAME #BASE,POINT2[] " ",TQ_STATE FALSE}
DECL E6POS XP296={X 1072.98704,Y -565.20086,Z 1272.32348,A -180,B 0,C 180,S 2,T 35,E1 0,E2 0,E3 0,E4 0,E5 0,E6 0}
; DECL LDAT LCPDATP42={VEL 1,ACC 100,APO_DIST 100,APO_FAC 50.0,ORI_TYP #VAR,CIRC_TYP #BASE,JERK_FAC 50.0}
DECL FDAT FP297={TOOL_NO 1,BASE_NO 2,IPO_FRAME #BASE,POINT2[] " ",TQ_STATE FALSE}
DECL E6POS XP297={X 1072.98689,Y -565.20116,Z 1122.32295,A 180,B 0,C -180,S 2,T 35,E1 0,E2 0,E3 0,E4 0,E5 0,E6 0}
; DECL LDAT LCPDATP43={VEL 1,ACC 100,APO_DIST 100,APO_FAC 50.0,ORI_TYP #VAR,CIRC_TYP #BASE,JERK_FAC 50.0}
DECL FDAT FP298={TOOL_NO 1,BASE_NO 2,IPO_FRAME #BASE,POINT2[] " ",TQ_STATE FALSE}
DECL E6POS XP298={X 1172.98673,Y -565.20078,Z 872.32277,A 180,B 0,C -180,S 2,T 35,E1 0,E2 0,E3 0,E4 0,E5 0,E6 0}
; DECL PDAT PPDATP23={VEL 100,ACC 100,APO_DIST 100,APO_MODE #CDIS,GEAR_JERK 100.000,EXAX_IGN 0}
DECL FDAT FP299={TOOL_NO 1,BASE_NO 2,IPO_FRAME #BASE,POINT2[] " ",TQ_STATE FALSE}
DECL E6POS XP299={X 681.98602,Y -565.20088,Z 1272.32295,A 180,B 0,C -180,S 2,T 35,E1 0,E2 0,E3 0,E4 0,E5 0,E6 0}
; DECL LDAT LCPDATP45={VEL 1,ACC 100,APO_DIST 100,APO_FAC 50.0,ORI_TYP #VAR,CIRC_TYP #BASE,JERK_FAC 50.0}
DECL FDAT FP300={TOOL_NO 1,BASE_NO 2,IPO_FRAME #BASE,POINT2[] " ",TQ_STATE FALSE}
DECL E6POS XP300={X 681.98616,Y -565.20081,Z 1122.3233,A -180,B 0,C -180,S 2,T 35,E1 0,E2 0,E3 0,E4 0,E5 0,E6 0}
; DECL LDAT LCPDATP44={VEL 1,ACC 100,APO_DIST 100,APO_FAC 50.0,ORI_TYP #VAR,CIRC_TYP #BASE,JERK_FAC 50.0}
DECL FDAT FP301={TOOL_NO 1,BASE_NO 2,IPO_FRAME #BASE,POINT2[] " ",TQ_STATE FALSE}
DECL E6POS XP301={X 781.9869,Y -565.20077,Z 872.32219,A 180,B 0,C 180,S 2,T 35,E1 0,E2 0,E3 0,E4 0,E5 0,E6 0}
; DECL PDAT PPDATP24={VEL 100,ACC 100,APO_DIST 100,APO_MODE #CDIS,GEAR_JERK 100.000,EXAX_IGN 0}
DECL FDAT FP302={TOOL_NO 1,BASE_NO 2,IPO_FRAME #BASE,POINT2[] " ",TQ_STATE FALSE}
DECL E6POS XP302={X 290.98722,Y -565.20115,Z 1272.32355,A 180,B 0,C -180,S 2,T 35,E1 0,E2 0,E3 0,E4 0,E5 0,E6 0}
; DECL LDAT LCPDATP46={VEL 1,ACC 100,APO_DIST 100,APO_FAC 50.0,ORI_TYP #VAR,CIRC_TYP #BASE,JERK_FAC 50.0}
DECL FDAT FP639={TOOL_NO 1,BASE_NO 2,IPO_FRAME #BASE,POINT2[] " ",TQ_STATE FALSE}
DECL E6POS XP639={X 290.9867,Y -565.20113,Z 1122.32278,A 180,B 0,C 180,S 2,T 35,E1 0,E2 0,E3 0,E4 0,E5 0,E6 0}
; DECL LDAT LCPDATP47={VEL 1,ACC 100,APO_DIST 100,APO_FAC 50.0,ORI_TYP #VAR,CIRC_TYP #BASE,JERK_FAC 50.0}
DECL FDAT FP640={TOOL_NO 1,BASE_NO 2,IPO_FRAME #BASE,POINT2[] " ",TQ_STATE FALSE}
DECL E6POS XP640={X 390.98701,Y -565.20118,Z 872.32277,A 180,B 0,C 180,S 2,T 35,E1 0,E2 0,E3 0,E4 0,E5 0,E6 0}
; ENDDAT for Mtrz_P2_32BarPacking
; Data for Pick_E_2_P_2_3
; DECL PDAT PPDATP1={VEL 100,ACC 100,APO_DIST 100,APO_MODE #CDIS,GEAR_JERK 100.000,EXAX_IGN 0}
DECL FDAT FP650={TOOL_NO 1,BASE_NO 4,IPO_FRAME #BASE,POINT2[] " ",TQ_STATE FALSE}
DECL E6POS XP650={X 542.90832,Y 2.83173,Z 2105.80063,A -90,B 0,C 180,S 2,T 3,E1 0,E2 0,E3 0,E4 0,E5 0,E6 0}
; DECL LDAT LCPDATP2={VEL 1,ACC 100,APO_DIST 100,APO_FAC 50.0,ORI_TYP #VAR,CIRC_TYP #BASE,JERK_FAC 50.0}
DECL FDAT FP651={TOOL_NO 1,BASE_NO 4,IPO_FRAME #BASE,POINT2[] " ",TQ_STATE FALSE}
DECL E6POS XP651={X 542.90832,Y 2.83193,Z 1391.79999,A -90,B 0,C -180,S 2,T 3,E1 0,E2 0,E3 0,E4 0,E5 0,E6 0}
; DECL LDAT LCPDATP1={VEL 1,ACC 100,APO_DIST 100,APO_FAC 50.0,ORI_TYP #VAR,CIRC_TYP #BASE,JERK_FAC 50.0}
DECL FDAT FPick_E_2_P_2_3={TOOL_NO 1,BASE_NO 4,IPO_FRAME #BASE,POINT2[] " ",TQ_STATE FALSE}
DECL E6POS XPick_E_2_P_2_3={X 542.90832,Y -19.40194,Z 1391.79999,A -90,B 0,C 180,S 2,T 3,E1 0,E2 0,E3 0,E4 0,E5 0,E6 0}
; DECL LDAT LCPDATP3={VEL 1,ACC 100,APO_DIST 100,APO_FAC 50.0,ORI_TYP #VAR,CIRC_TYP #BASE,JERK_FAC 50.0}
DECL FDAT FP652={TOOL_NO 1,BASE_NO 4,IPO_FRAME #BASE,POINT2[] " ",TQ_STATE FALSE}
DECL E6POS XP652={X 542.90832,Y -19.40201,Z 2105.79999,A -90,B 0,C -180,S 2,T 3,E1 0,E2 0,E3 0,E4 0,E5 0,E6 0}
; ENDDAT for Pick_E_2_P_2_3
; Data for Mtrz_P2_33BarPacking
; DECL PDAT PPDATP25={VEL 100,ACC 100,APO_DIST 100,APO_MODE #CDIS,GEAR_JERK 100.000,EXAX_IGN 0}
DECL FDAT FP653={TOOL_NO 1,BASE_NO 2,IPO_FRAME #BASE,POINT2[] " ",TQ_STATE FALSE}
DECL E6POS XP653={X 1047.81428,Y -532.63231,Z 1263.51475,A 180,B 0,C 180,S 2,T 35,E1 0,E2 0,E3 0,E4 0,E5 0,E6 0}
; DECL LDAT LCPDATP48={VEL 1,ACC 100,APO_DIST 100,APO_FAC 50.0,ORI_TYP #VAR,CIRC_TYP #BASE,JERK_FAC 50.0}
DECL FDAT FP654={TOOL_NO 1,BASE_NO 2,IPO_FRAME #BASE,POINT2[] " ",TQ_STATE FALSE}
DECL E6POS XP654={X 1047.81429,Y -532.63247,Z 1063.51485,A 180,B 0,C 180,S 2,T 35,E1 0,E2 0,E3 0,E4 0,E5 0,E6 0}
; DECL LDAT LCPDATP49={VEL 1,ACC 100,APO_DIST 100,APO_FAC 50.0,ORI_TYP #VAR,CIRC_TYP #BASE,JERK_FAC 50.0}
DECL FDAT FP655={TOOL_NO 1,BASE_NO 2,IPO_FRAME #BASE,POINT2[] " ",TQ_STATE FALSE}
DECL E6POS XP655={X 1147.81449,Y -532.63244,Z 863.51516,A 180,B 0,C 180,S 2,T 35,E1 0,E2 0,E3 0,E4 0,E5 0,E6 0}
; DECL PDAT PPDATP26={VEL 100,ACC 100,APO_DIST 100,APO_MODE #CDIS,GEAR_JERK 100.000,EXAX_IGN 0}
DECL FDAT FP656={TOOL_NO 1,BASE_NO 2,IPO_FRAME #BASE,POINT2[] " ",TQ_STATE FALSE}
DECL E6POS XP656={X 482.81525,Y -532.63229,Z 1263.51579,A 180,B 0,C 180,S 2,T 35,E1 0,E2 0,E3 0,E4 0,E5 0,E6 0}
; DECL LDAT LCPDATP50={VEL 1,ACC 100,APO_DIST 100,APO_FAC 50.0,ORI_TYP #VAR,CIRC_TYP #BASE,JERK_FAC 50.0}
DECL FDAT FP657={TOOL_NO 1,BASE_NO 2,IPO_FRAME #BASE,POINT2[] " ",TQ_STATE FALSE}
DECL E6POS XP657={X 482.81509,Y -532.63223,Z 1063.51535,A 180,B 0,C 180,S 2,T 35,E1 0,E2 0,E3 0,E4 0,E5 0,E6 0}
; DECL LDAT LCPDATP51={VEL 1,ACC 100,APO_DIST 100,APO_FAC 50.0,ORI_TYP #VAR,CIRC_TYP #BASE,JERK_FAC 50.0}
DECL FDAT FP658={TOOL_NO 1,BASE_NO 2,IPO_FRAME #BASE,POINT2[] " ",TQ_STATE FALSE}
DECL E6POS XP658={X 582.81489,Y -532.63218,Z 863.51495,A -180,B 0,C 180,S 2,T 35,E1 0,E2 0,E3 0,E4 0,E5 0,E6 0}
; ENDDAT for Mtrz_P2_33BarPacking
; Data for Mtrz_P2_34BarPacking
; DECL PDAT PPDATP27={VEL 100,ACC 100,APO_DIST 100,APO_MODE #CDIS,GEAR_JERK 100.000,EXAX_IGN 0}
DECL FDAT FP113={TOOL_NO 1,BASE_NO 2,IPO_FRAME #BASE,POINT2[] " ",TQ_STATE FALSE}
DECL E6POS XP113={X 1055.40866,Y -747.77738,Z 1006.97196,A -180,B 0,C -180,S 2,T 35,E1 0,E2 0,E3 0,E4 0,E5 0,E6 0}
; DECL LDAT LCPDATP52={VEL 1,ACC 100,APO_DIST 100,APO_FAC 50.0,ORI_TYP #VAR,CIRC_TYP #BASE,JERK_FAC 50.0}
DECL FDAT FP130={TOOL_NO 1,BASE_NO 2,IPO_FRAME #BASE,POINT2[] " ",TQ_STATE FALSE}
DECL E6POS XP130={X 1055.40912,Y -747.77793,Z 886.97188,A -180,B 0,C -180,S 2,T 35,E1 0,E2 0,E3 0,E4 0,E5 0,E6 0}
; DECL LDAT LCPDATP53={VEL 1,ACC 100,APO_DIST 100,APO_FAC 50.0,ORI_TYP #VAR,CIRC_TYP #BASE,JERK_FAC 50.0}
DECL FDAT FP131={TOOL_NO 1,BASE_NO 2,IPO_FRAME #BASE,POINT2[] " ",TQ_STATE FALSE}
DECL E6POS XP131={X 1155.40894,Y -747.77773,Z 786.97153,A -180,B 0,C 180,S 2,T 35,E1 0,E2 0,E3 0,E4 0,E5 0,E6 0}
; DECL PDAT PPDATP29={VEL 100,ACC 100,APO_DIST 100,APO_MODE #CDIS,GEAR_JERK 100.000,EXAX_IGN 0}
DECL FDAT FP132={TOOL_NO 1,BASE_NO 2,IPO_FRAME #BASE,POINT2[] " ",TQ_STATE FALSE}
DECL E6POS XP132={X 516.40798,Y -747.778,Z 1006.97252,A -180,B 0,C 180,S 2,T 35,E1 0,E2 0,E3 0,E4 0,E5 0,E6 0}
; DECL LDAT LCPDATP54={VEL 1,ACC 100,APO_DIST 100,APO_FAC 50.0,ORI_TYP #VAR,CIRC_TYP #BASE,JERK_FAC 50.0}
DECL FDAT FP133={TOOL_NO 1,BASE_NO 2,IPO_FRAME #BASE,POINT2[] " ",TQ_STATE FALSE}
DECL E6POS XP133={X 516.40827,Y -747.77795,Z 886.97211,A -180,B 0,C -180,S 2,T 35,E1 0,E2 0,E3 0,E4 0,E5 0,E6 0}
; DECL LDAT LCPDATP55={VEL 1,ACC 100,APO_DIST 100,APO_FAC 50.0,ORI_TYP #VAR,CIRC_TYP #BASE,JERK_FAC 50.0}
DECL FDAT FP202={TOOL_NO 1,BASE_NO 2,IPO_FRAME #BASE,POINT2[] " ",TQ_STATE FALSE}
DECL E6POS XP202={X 586.40852,Y -747.7776,Z 786.97168,A 180,B 0,C 180,S 2,T 35,E1 0,E2 0,E3 0,E4 0,E5 0,E6 0}
; ENDDAT for Mtrz_P2_34BarPacking
; Data for Pick_E_2_P_3
; DECL PDAT PPDATP1={VEL 100,ACC 100,APO_DIST 100,APO_MODE #CDIS,GEAR_JERK 100.000,EXAX_IGN 0}
DECL FDAT FP203={TOOL_NO 1,BASE_NO 4,IPO_FRAME #BASE,POINT2[] " ",TQ_STATE FALSE}
DECL E6POS XP203={X 484.9373,Y 0.60233,Z 2072.81668,A -90,B 0,C -180,S 2,T 3,E1 0,E2 0,E3 0,E4 0,E5 0,E6 0}
; DECL LDAT LCPDATP2={VEL 1,ACC 100,APO_DIST 100,APO_FAC 50.0,ORI_TYP #VAR,CIRC_TYP #BASE,JERK_FAC 50.0}
DECL FDAT FP204={TOOL_NO 1,BASE_NO 4,IPO_FRAME #BASE,POINT2[] " ",TQ_STATE FALSE}
DECL E6POS XP204={X 484.9373,Y 0.60122,Z 1393.78865,A -90,B 0,C -180,S 2,T 3,E1 0,E2 0,E3 0,E4 0,E5 0,E6 0}
; DECL LDAT LCPDATP1={VEL 1,ACC 100,APO_DIST 100,APO_FAC 50.0,ORI_TYP #VAR,CIRC_TYP #BASE,JERK_FAC 50.0}
DECL FDAT FPick_E_2_P_3={TOOL_NO 1,BASE_NO 4,IPO_FRAME #BASE,POINT2[] " ",TQ_STATE FALSE}
DECL E6POS XPick_E_2_P_3={X 484.9373,Y -56.83179,Z 1342.79999,A -90,B 0,C -180,S 2,T 3,E1 0,E2 0,E3 0,E4 0,E5 0,E6 0}
; DECL LDAT LCPDATP3={VEL 1,ACC 100,APO_DIST 100,APO_FAC 50.0,ORI_TYP #VAR,CIRC_TYP #BASE,JERK_FAC 50.0}
DECL FDAT FP205={TOOL_NO 1,BASE_NO 4,IPO_FRAME #BASE,POINT2[] " ",TQ_STATE FALSE}
DECL E6POS XP205={X 484.9373,Y -56.83191,Z 2072.81819,A -90,B 0,C 180,S 2,T 3,E1 0,E2 0,E3 0,E4 0,E5 0,E6 0}
; ENDDAT for Pick_E_2_P_3
; Data for Mtrz_P2_9Aero
; DECL PDAT PPDATP5={VEL 100,ACC 100,APO_DIST 100,APO_MODE #CDIS,GEAR_JERK 100.000,EXAX_IGN 0}
DECL FDAT FP72={TOOL_NO 1,BASE_NO 2,IPO_FRAME #BASE,POINT2[] " ",TQ_STATE FALSE}
DECL E6POS XP72={X 1022.73266,Y -478.76887,Z 1036.99508,A -180,B 0,C 180,S 2,T 35,E1 0,E2 0,E3 0,E4 0,E5 0,E6 0}
; DECL LDAT LCPDATP98={VEL 1,ACC 100,APO_DIST 100,APO_FAC 50.0,ORI_TYP #VAR,CIRC_TYP #BASE,JERK_FAC 50.0}
DECL FDAT FP659={TOOL_NO 1,BASE_NO 2,IPO_FRAME #BASE,POINT2[] " ",TQ_STATE FALSE}
DECL E6POS XP659={X 1022.73295,Y -478.7684,Z 936.99495,A 180,B 0,C 180,S 2,T 35,E1 0,E2 0,E3 0,E4 0,E5 0,E6 0}
; DECL LDAT LCPDATP99={VEL 1,ACC 100,APO_DIST 100,APO_FAC 50.0,ORI_TYP #VAR,CIRC_TYP #BASE,JERK_FAC 50.0}
DECL FDAT FP660={TOOL_NO 1,BASE_NO 2,IPO_FRAME #BASE,POINT2[] " ",TQ_STATE FALSE}
DECL E6POS XP660={X 1122.73281,Y -478.76864,Z 786.99517,A -180,B 0,C -180,S 2,T 35,E1 0,E2 0,E3 0,E4 0,E5 0,E6 0}
; DECL PDAT PPDATP50={VEL 100,ACC 100,APO_DIST 100,APO_MODE #CDIS,GEAR_JERK 100.000,EXAX_IGN 0}
DECL FDAT FP661={TOOL_NO 1,BASE_NO 2,IPO_FRAME #BASE,POINT2[] " ",TQ_STATE FALSE}
DECL E6POS XP661={X 536.73268,Y -478.76855,Z 1036.99478,A -180,B 0,C 180,S 2,T 35,E1 0,E2 0,E3 0,E4 0,E5 0,E6 0}
; DECL LDAT LCPDATP100={VEL 1,ACC 100,APO_DIST 100,APO_FAC 50.0,ORI_TYP #VAR,CIRC_TYP #BASE,JERK_FAC 50.0}
DECL FDAT FP662={TOOL_NO 1,BASE_NO 2,IPO_FRAME #BASE,POINT2[] " ",TQ_STATE FALSE}
DECL E6POS XP662={X 536.73295,Y -478.76869,Z 936.99466,A -180,B 0,C -180,S 2,T 35,E1 0,E2 0,E3 0,E4 0,E5 0,E6 0}
; DECL LDAT LCPDATP101={VEL 1,ACC 100,APO_DIST 100,APO_FAC 50.0,ORI_TYP #VAR,CIRC_TYP #BASE,JERK_FAC 50.0}
DECL FDAT FP663={TOOL_NO 1,BASE_NO 2,IPO_FRAME #BASE,POINT2[] " ",TQ_STATE FALSE}
DECL E6POS XP663={X 586.73291,Y -478.76888,Z 786.99521,A 180,B 0,C -180,S 2,T 35,E1 0,E2 0,E3 0,E4 0,E5 0,E6 0}
; ENDDAT for Mtrz_P2_9Aero
; Data for Mtrz_P2_23Smarties
; DECL PDAT PPDATP79={VEL 100,ACC 100,APO_DIST 100,APO_MODE #CDIS,GEAR_JERK 100.000,EXAX_IGN 0}
DECL FDAT FP393={TOOL_NO 1,BASE_NO 2,IPO_FRAME #BASE,POINT2[] " ",TQ_STATE FALSE}
DECL E6POS XP393={X 680.29786,Y -46.52966,Z 1158.21795,A -90,B 0,C 180,S 2,T 35,E1 0,E2 0,E3 0,E4 0,E5 0,E6 0}
; DECL LDAT LCPDATP159={VEL 1,ACC 100,APO_DIST 100,APO_FAC 50.0,ORI_TYP #VAR,CIRC_TYP #BASE,JERK_FAC 50.0}
DECL FDAT FP425={TOOL_NO 1,BASE_NO 2,IPO_FRAME #BASE,POINT2[] " ",TQ_STATE FALSE}
DECL E6POS XP425={X 680.29815,Y -46.52974,Z 958.21648,A -90,B 0,C 180,S 2,T 35,E1 0,E2 0,E3 0,E4 0,E5 0,E6 0}
; DECL LDAT LCPDATP158={VEL 1,ACC 100,APO_DIST 100,APO_FAC 50.0,ORI_TYP #VAR,CIRC_TYP #BASE,JERK_FAC 50.0}
DECL FDAT FP670={TOOL_NO 1,BASE_NO 2,IPO_FRAME #BASE,POINT2[] " ",TQ_STATE FALSE}
DECL E6POS XP670={X 730.29868,Y 3.47028,Z 858.21742,A -90,B 0,C 180,S 2,T 35,E1 0,E2 0,E3 0,E4 0,E5 0,E6 0}
; DECL PDAT PPDATP80={VEL 100,ACC 100,APO_DIST 100,APO_MODE #CDIS,GEAR_JERK 100.000,EXAX_IGN 0}
DECL FDAT FP671={TOOL_NO 1,BASE_NO 2,IPO_FRAME #BASE,POINT2[] " ",TQ_STATE FALSE}
DECL E6POS XP671={X 220.31123,Y -45.53425,Z 1162.94486,A -90,B 0,C 180,S 2,T 35,E1 0,E2 0,E3 0,E4 0,E5 0,E6 0}
; DECL LDAT LCPDATP161={VEL 1,ACC 100,APO_DIST 100,APO_FAC 50.0,ORI_TYP #VAR,CIRC_TYP #BASE,JERK_FAC 50.0}
DECL FDAT FP672={TOOL_NO 1,BASE_NO 2,IPO_FRAME #BASE,POINT2[] " ",TQ_STATE FALSE}
DECL E6POS XP672={X 220.31125,Y -45.53425,Z 958.21844,A -90,B 0,C 180,S 2,T 35,E1 0,E2 0,E3 0,E4 0,E5 0,E6 0}
; DECL LDAT LCPDATP160={VEL 1,ACC 100,APO_DIST 100,APO_FAC 50.0,ORI_TYP #VAR,CIRC_TYP #BASE,JERK_FAC 50.0}
DECL FDAT FP673={TOOL_NO 1,BASE_NO 2,IPO_FRAME #BASE,POINT2[] " ",TQ_STATE FALSE}
DECL E6POS XP673={X 260.31117,Y 3.46852,Z 858.20469,A -90,B 0,C 180,S 2,T 35,E1 0,E2 0,E3 0,E4 0,E5 0,E6 0}
; DECL PDAT PPDATP81={VEL 100,ACC 100,APO_DIST 100,APO_MODE #CDIS,GEAR_JERK 100.000,EXAX_IGN 0}
DECL FDAT FP674={TOOL_NO 1,BASE_NO 2,IPO_FRAME #BASE,POINT2[] " ",TQ_STATE FALSE}
DECL E6POS XP674={X 730.3109,Y -550.52888,Z 1158.21899,A -90,B 0,C 180,S 2,T 35,E1 0,E2 0,E3 0,E4 0,E5 0,E6 0}
; DECL LDAT LCPDATP163={VEL 1,ACC 100,APO_DIST 100,APO_FAC 50.0,ORI_TYP #VAR,CIRC_TYP #BASE,JERK_FAC 50.0}
DECL FDAT FP675={TOOL_NO 1,BASE_NO 2,IPO_FRAME #BASE,POINT2[] " ",TQ_STATE FALSE}
DECL E6POS XP675={X 730.31094,Y -550.52948,Z 958.21714,A -90,B 0,C 180,S 2,T 35,E1 0,E2 0,E3 0,E4 0,E5 0,E6 0}
; DECL LDAT LCPDATP162={VEL 1,ACC 100,APO_DIST 100,APO_FAC 50.0,ORI_TYP #VAR,CIRC_TYP #BASE,JERK_FAC 50.0}
DECL FDAT FP676={TOOL_NO 1,BASE_NO 2,IPO_FRAME #BASE,POINT2[] " ",TQ_STATE FALSE}
DECL E6POS XP676={X 730.31175,Y -500.53121,Z 858.20394,A -90,B 0,C 180,S 2,T 35,E1 0,E2 0,E3 0,E4 0,E5 0,E6 0}
; DECL PDAT PPDATP82={VEL 100,ACC 100,APO_DIST 100,APO_MODE #CDIS,GEAR_JERK 100.000,EXAX_IGN 0}
DECL FDAT FP677={TOOL_NO 1,BASE_NO 2,IPO_FRAME #BASE,POINT2[] " ",TQ_STATE FALSE}
DECL E6POS XP677={X 220.31162,Y -549.53479,Z 1140.51232,A -90,B 0,C 180,S 2,T 35,E1 0,E2 0,E3 0,E4 0,E5 0,E6 0}
; DECL LDAT LCPDATP165={VEL 1,ACC 100,APO_DIST 100,APO_FAC 50.0,ORI_TYP #VAR,CIRC_TYP #BASE,JERK_FAC 50.0}
DECL FDAT FP678={TOOL_NO 1,BASE_NO 2,IPO_FRAME #BASE,POINT2[] " ",TQ_STATE FALSE}
DECL E6POS XP678={X 220.31152,Y -549.5345,Z 958.21889,A -90,B 0,C 180,S 2,T 35,E1 0,E2 0,E3 0,E4 0,E5 0,E6 0}
; DECL LDAT LCPDATP164={VEL 1,ACC 100,APO_DIST 100,APO_FAC 50.0,ORI_TYP #VAR,CIRC_TYP #BASE,JERK_FAC 50.0}
DECL FDAT FP679={TOOL_NO 1,BASE_NO 2,IPO_FRAME #BASE,POINT2[] " ",TQ_STATE FALSE}
DECL E6POS XP679={X 260.31142,Y -500.53004,Z 858.20277,A -90,B 0,C -180,S 2,T 35,E1 0,E2 0,E3 0,E4 0,E5 0,E6 0}
DECL PDAT PPDATP89={VEL 100,ACC 100,APO_DIST 100,APO_MODE #CDIS,GEAR_JERK 100.000,EXAX_IGN 0}
DECL FDAT FP75={TOOL_NO 1,BASE_NO 2,IPO_FRAME #BASE,POINT2[] " ",TQ_STATE FALSE}
DECL E6POS XP75={X 561.19813,Y -57.20487,Z 1363.2041,A -90,B 0,C 180,S 2,T 35,E1 0,E2 0,E3 0,E4 0,E5 0,E6 0}
DECL LDAT LCPDATP177={VEL 1,ACC 100,APO_DIST 100,APO_FAC 50.0,ORI_TYP #VAR,CIRC_TYP #BASE,JERK_FAC 50.0}
DECL FDAT FP74={TOOL_NO 1,BASE_NO 2,IPO_FRAME #BASE,POINT2[] " ",TQ_STATE FALSE}
DECL E6POS XP74={X 561.19825,Y -57.20482,Z 1213.2044,A -90,B 0,C 180,S 2,T 35,E1 0,E2 0,E3 0,E4 0,E5 0,E6 0}
DECL LDAT LCPDATP176={VEL 1,ACC 100,APO_DIST 100,APO_FAC 50.0,ORI_TYP #VAR,CIRC_TYP #BASE,JERK_FAC 50.0}
DECL FDAT FP73={TOOL_NO 1,BASE_NO 2,IPO_FRAME #BASE,POINT2[] " ",TQ_STATE FALSE}
DECL E6POS XP73={X 511.19825,Y -7.20482,Z 1113.20441,A -90,B 0,C 180,S 2,T 35,E1 0,E2 0,E3 0,E4 0,E5 0,E6 0}
; DECL PDAT PPDATP83={VEL 100,ACC 100,APO_DIST 100,APO_MODE #CDIS,GEAR_JERK 100.000,EXAX_IGN 0}
DECL FDAT FP683={TOOL_NO 1,BASE_NO 2,IPO_FRAME #BASE,POINT2[] " ",TQ_STATE FALSE}
DECL E6POS XP683={X 1021.20299,Y -49.72447,Z 1413.21833,A -90,B 0,C 180,S 2,T 3,E1 0,E2 0,E3 0,E4 0,E5 0,E6 0}
; DECL LDAT LCPDATP167={VEL 1,ACC 100,APO_DIST 100,APO_FAC 50.0,ORI_TYP #VAR,CIRC_TYP #BASE,JERK_FAC 50.0}
DECL FDAT FP684={TOOL_NO 1,BASE_NO 2,IPO_FRAME #BASE,POINT2[] " ",TQ_STATE FALSE}
DECL E6POS XP684={X 1021.20299,Y -49.72454,Z 1213.21653,A -90,B 0,C 180,S 2,T 3,E1 0,E2 0,E3 0,E4 0,E5 0,E6 0}
; DECL LDAT LCPDATP166={VEL 1,ACC 100,APO_DIST 100,APO_FAC 50.0,ORI_TYP #VAR,CIRC_TYP #BASE,JERK_FAC 50.0}
DECL FDAT FP685={TOOL_NO 1,BASE_NO 2,IPO_FRAME #BASE,POINT2[] " ",TQ_STATE FALSE}
DECL E6POS XP685={X 981.20299,Y -7.19653,Z 1113.21365,A -90,B 0,C 180,S 2,T 3,E1 0,E2 0,E3 0,E4 0,E5 0,E6 0}
; DECL PDAT PPDATP83={VEL 100,ACC 100,APO_DIST 100,APO_MODE #CDIS,GEAR_JERK 100.000,EXAX_IGN 0}
DECL FDAT FP686={TOOL_NO 1,BASE_NO 2,IPO_FRAME #BASE,POINT2[] " ",TQ_STATE FALSE}
DECL E6POS XP686={X 561.19928,Y -593.72483,Z 1413.21893,A -90,B 0,C 180,S 2,T 35,E1 0,E2 0,E3 0,E4 0,E5 0,E6 0}
; DECL LDAT LCPDATP167={VEL 1,ACC 100,APO_DIST 100,APO_FAC 50.0,ORI_TYP #VAR,CIRC_TYP #BASE,JERK_FAC 50.0}
DECL FDAT FP687={TOOL_NO 1,BASE_NO 2,IPO_FRAME #BASE,POINT2[] " ",TQ_STATE FALSE}
DECL E6POS XP687={X 561.19963,Y -593.72483,Z 1213.21659,A -90,B 0,C 180,S 2,T 35,E1 0,E2 0,E3 0,E4 0,E5 0,E6 0}
; DECL LDAT LCPDATP166={VEL 1,ACC 100,APO_DIST 100,APO_FAC 50.0,ORI_TYP #VAR,CIRC_TYP #BASE,JERK_FAC 50.0}
DECL FDAT FP688={TOOL_NO 1,BASE_NO 2,IPO_FRAME #BASE,POINT2[] " ",TQ_STATE FALSE}
DECL E6POS XP688={X 511.19963,Y -511.20495,Z 1113.20485,A -90,B 0,C 180,S 2,T 35,E1 0,E2 0,E3 0,E4 0,E5 0,E6 0}
; DECL PDAT PPDATP83={VEL 100,ACC 100,APO_DIST 100,APO_MODE #CDIS,GEAR_JERK 100.000,EXAX_IGN 0}
DECL FDAT FP689={TOOL_NO 1,BASE_NO 2,IPO_FRAME #BASE,POINT2[] " ",TQ_STATE FALSE}
DECL E6POS XP689={X 1031.20332,Y -593.7245,Z 1413.21869,A -90,B 0,C 180,S 2,T 3,E1 0,E2 0,E3 0,E4 0,E5 0,E6 0}
; DECL LDAT LCPDATP167={VEL 1,ACC 100,APO_DIST 100,APO_FAC 50.0,ORI_TYP #VAR,CIRC_TYP #BASE,JERK_FAC 50.0}
DECL FDAT FP690={TOOL_NO 1,BASE_NO 2,IPO_FRAME #BASE,POINT2[] " ",TQ_STATE FALSE}
DECL E6POS XP690={X 1031.20318,Y -593.7245,Z 1213.21651,A -90,B 0,C 180,S 2,T 3,E1 0,E2 0,E3 0,E4 0,E5 0,E6 0}
; DECL LDAT LCPDATP166={VEL 1,ACC 100,APO_DIST 100,APO_FAC 50.0,ORI_TYP #VAR,CIRC_TYP #BASE,JERK_FAC 50.0}
DECL FDAT FP691={TOOL_NO 1,BASE_NO 2,IPO_FRAME #BASE,POINT2[] " ",TQ_STATE FALSE}
DECL E6POS XP691={X 981.20318,Y -511.19805,Z 1113.21157,A -90,B 0,C 180,S 2,T 3,E1 0,E2 0,E3 0,E4 0,E5 0,E6 0}
; ENDDAT for Mtrz_P2_23Smarties
; Data for Pick_E_2_P_4
; DECL PDAT PPDATP1={VEL 100,ACC 100,APO_DIST 100,APO_MODE #CDIS,GEAR_JERK 100.000,EXAX_IGN 0}
DECL FDAT FP692={TOOL_NO 1,BASE_NO 4,IPO_FRAME #BASE,POINT2[] " ",TQ_STATE FALSE}
DECL E6POS XP692={X 465.93753,Y -572.77244,Z 2072.81751,A 90,B 0,C -180,S 2,T 3,E1 0,E2 0,E3 0,E4 0,E5 0,E6 0}
; DECL LDAT LCPDATP2={VEL 1,ACC 100,APO_DIST 100,APO_FAC 50.0,ORI_TYP #VAR,CIRC_TYP #BASE,JERK_FAC 50.0}
DECL FDAT FP693={TOOL_NO 1,BASE_NO 4,IPO_FRAME #BASE,POINT2[] " ",TQ_STATE FALSE}
DECL E6POS XP693={X 465.9373,Y -572.77204,Z 1354.26523,A 90,B 0,C 180,S 2,T 3,E1 0,E2 0,E3 0,E4 0,E5 0,E6 0}
; DECL LDAT LCPDATP1={VEL 1,ACC 100,APO_DIST 100,APO_FAC 50.0,ORI_TYP #VAR,CIRC_TYP #BASE,JERK_FAC 50.0}
DECL FDAT FPick_E_2_P_4={TOOL_NO 1,BASE_NO 4,IPO_FRAME #BASE,POINT2[] " ",TQ_STATE FALSE}
DECL E6POS XPick_E_2_P_4={X 465.9373,Y -502.13378,Z 1391.79999,A 90,B 0,C 180,S 2,T 3,E1 0,E2 0,E3 0,E4 0,E5 0,E6 0}
; DECL LDAT LCPDATP3={VEL 1,ACC 100,APO_DIST 100,APO_FAC 50.0,ORI_TYP #VAR,CIRC_TYP #BASE,JERK_FAC 50.0}
DECL FDAT FP694={TOOL_NO 1,BASE_NO 4,IPO_FRAME #BASE,POINT2[] " ",TQ_STATE FALSE}
DECL E6POS XP694={X 465.9373,Y -502.13386,Z 2072.81818,A 90,B 0,C 180,S 2,T 3,E1 0,E2 0,E3 0,E4 0,E5 0,E6 0}
; ENDDAT for Pick_E_2_P_4
; Data for Pick_E_2_P_5
; DECL PDAT PPDATP1={VEL 100,ACC 100,APO_DIST 100,APO_MODE #CDIS,GEAR_JERK 100.000,EXAX_IGN 0}
DECL FDAT FP695={TOOL_NO 1,BASE_NO 4,IPO_FRAME #BASE,POINT2[] " ",TQ_STATE FALSE}
DECL E6POS XP695={X 482.9373,Y 2.8323,Z 2072.81708,A -90,B 0,C -180,S 2,T 3,E1 0,E2 0,E3 0,E4 0,E5 0,E6 0}
; DECL LDAT LCPDATP2={VEL 1,ACC 100,APO_DIST 100,APO_FAC 50.0,ORI_TYP #VAR,CIRC_TYP #BASE,JERK_FAC 50.0}
DECL FDAT FP696={TOOL_NO 1,BASE_NO 4,IPO_FRAME #BASE,POINT2[] " ",TQ_STATE FALSE}
DECL E6POS XP696={X 482.9373,Y 2.83181,Z 1359.49624,A -90,B 0,C -180,S 2,T 3,E1 0,E2 0,E3 0,E4 0,E5 0,E6 0}
; DECL LDAT LCPDATP1={VEL 1,ACC 100,APO_DIST 100,APO_FAC 50.0,ORI_TYP #VAR,CIRC_TYP #BASE,JERK_FAC 50.0}
DECL FDAT FPick_E_2_P_5={TOOL_NO 1,BASE_NO 4,IPO_FRAME #BASE,POINT2[] " ",TQ_STATE FALSE}
DECL E6POS XPick_E_2_P_5={X 482.9373,Y -19.40188,Z 1391.79999,A -90,B 0,C -180,S 2,T 3,E1 0,E2 0,E3 0,E4 0,E5 0,E6 0}
; DECL LDAT LCPDATP3={VEL 1,ACC 100,APO_DIST 100,APO_FAC 50.0,ORI_TYP #VAR,CIRC_TYP #BASE,JERK_FAC 50.0}
DECL FDAT FP697={TOOL_NO 1,BASE_NO 4,IPO_FRAME #BASE,POINT2[] " ",TQ_STATE FALSE}
DECL E6POS XP697={X 482.9373,Y -19.40183,Z 2072.81804,A -90,B 0,C -180,S 2,T 3,E1 0,E2 0,E3 0,E4 0,E5 0,E6 0}
; ENDDAT for Pick_E_2_P_5
; Data for Mtrz_P2_10CoffeCrisp
; DECL PDAT PPDATP56={VEL 100,ACC 100,APO_DIST 100,APO_MODE #CDIS,GEAR_JERK 100.000,EXAX_IGN 0}
DECL FDAT FP258={TOOL_NO 1,BASE_NO 2,IPO_FRAME #BASE,POINT2[] " ",TQ_STATE FALSE}
DECL E6POS XP258={X 678.68703,Y -69.47041,Z 1064.60184,A -90,B 0,C 180,S 2,T 35,E1 0,E2 0,E3 0,E4 0,E5 0,E6 0}
; DECL LDAT LCPDATP118={VEL 1,ACC 100,APO_DIST 100,APO_FAC 50.0,ORI_TYP #VAR,CIRC_TYP #BASE,JERK_FAC 50.0}
DECL FDAT FP259={TOOL_NO 1,BASE_NO 2,IPO_FRAME #BASE,POINT2[] " ",TQ_STATE FALSE}
DECL E6POS XP259={X 678.68701,Y -69.47031,Z 964.6022,A -90,B 0,C 180,S 2,T 35,E1 0,E2 0,E3 0,E4 0,E5 0,E6 0}
; DECL LDAT LCPDATP119={VEL 1,ACC 100,APO_DIST 100,APO_FAC 50.0,ORI_TYP #VAR,CIRC_TYP #BASE,JERK_FAC 50.0}
DECL FDAT FP260={TOOL_NO 1,BASE_NO 2,IPO_FRAME #BASE,POINT2[] " ",TQ_STATE FALSE}
DECL E6POS XP260={X 678.68718,Y 30.52967,Z 814.6017,A -90,B 0,C 180,S 2,T 35,E1 0,E2 0,E3 0,E4 0,E5 0,E6 0}
; DECL PDAT PPDATP60={VEL 100,ACC 100,APO_DIST 100,APO_MODE #CDIS,GEAR_JERK 100.000,EXAX_IGN 0}
DECL FDAT FP261={TOOL_NO 1,BASE_NO 2,IPO_FRAME #BASE,POINT2[] " ",TQ_STATE FALSE}
DECL E6POS XP261={X 678.68644,Y -549.47075,Z 1064.60202,A -90,B 0,C 180,S 2,T 35,E1 0,E2 0,E3 0,E4 0,E5 0,E6 0}
; DECL LDAT LCPDATP121={VEL 1,ACC 100,APO_DIST 100,APO_FAC 50.0,ORI_TYP #VAR,CIRC_TYP #BASE,JERK_FAC 50.0}
DECL FDAT FP262={TOOL_NO 1,BASE_NO 2,IPO_FRAME #BASE,POINT2[] " ",TQ_STATE FALSE}
DECL E6POS XP262={X 678.68631,Y -549.47009,Z 964.60168,A -90,B 0,C 180,S 2,T 35,E1 0,E2 0,E3 0,E4 0,E5 0,E6 0}
; DECL LDAT LCPDATP120={VEL 1,ACC 100,APO_DIST 100,APO_FAC 50.0,ORI_TYP #VAR,CIRC_TYP #BASE,JERK_FAC 50.0}
DECL FDAT FP263={TOOL_NO 1,BASE_NO 2,IPO_FRAME #BASE,POINT2[] " ",TQ_STATE FALSE}
DECL E6POS XP263={X 678.68613,Y -449.47014,Z 814.60185,A -90,B 0,C 180,S 2,T 35,E1 0,E2 0,E3 0,E4 0,E5 0,E6 0}
DECL PDAT PPDATP90={VEL 100,ACC 100,APO_DIST 100,APO_MODE #CDIS,GEAR_JERK 100.000,EXAX_IGN 0}
DECL FDAT FP89={TOOL_NO 1,BASE_NO 2,IPO_FRAME #BASE,POINT2[] " ",TQ_STATE FALSE}
DECL E6POS XP89={X 916.04623,Y -625.2762,Z 1065.37648,A -180,B 0,C 180,S 2,T 35,E1 0,E2 0,E3 0,E4 0,E5 0,E6 0}
; DECL LDAT LCPDATP122={VEL 1,ACC 100,APO_DIST 100,APO_FAC 50.0,ORI_TYP #VAR,CIRC_TYP #BASE,JERK_FAC 50.0}
DECL FDAT FP265={TOOL_NO 1,BASE_NO 2,IPO_FRAME #BASE,POINT2[] " ",TQ_STATE FALSE}
DECL E6POS XP265={X 916.04603,Y -625.27628,Z 915.37674,A -180,B 0,C 180,S 2,T 35,E1 0,E2 0,E3 0,E4 0,E5 0,E6 0}
; DECL LDAT LCPDATP123={VEL 1,ACC 100,APO_DIST 100,APO_FAC 50.0,ORI_TYP #VAR,CIRC_TYP #BASE,JERK_FAC 50.0}
DECL FDAT FP266={TOOL_NO 1,BASE_NO 2,IPO_FRAME #BASE,POINT2[] " ",TQ_STATE FALSE}
DECL E6POS XP266={X 966.04643,Y -625.27632,Z 815.37641,A -180,B 0,C 180,S 2,T 35,E1 0,E2 0,E3 0,E4 0,E5 0,E6 0}
DECL PDAT PPDATP91={VEL 100,ACC 100,APO_DIST 100,APO_MODE #CDIS,GEAR_JERK 100.000,EXAX_IGN 0}
DECL FDAT FP90={TOOL_NO 1,BASE_NO 2,IPO_FRAME #BASE,POINT2[] " ",TQ_STATE FALSE}
DECL E6POS XP90={X 451.05208,Y -625.2666,Z 1065.37634,A 180,B 0,C 180,S 2,T 35,E1 0,E2 0,E3 0,E4 0,E5 0,E6 0}
; DECL LDAT LCPDATP125={VEL 1,ACC 100,APO_DIST 100,APO_FAC 50.0,ORI_TYP #VAR,CIRC_TYP #BASE,JERK_FAC 50.0}
DECL FDAT FP268={TOOL_NO 1,BASE_NO 2,IPO_FRAME #BASE,POINT2[] " ",TQ_STATE FALSE}
DECL E6POS XP268={X 451.05203,Y -625.26648,Z 915.36233,A -180,B 0,C -180,S 2,T 35,E1 0,E2 0,E3 0,E4 0,E5 0,E6 0}
; DECL LDAT LCPDATP124={VEL 1,ACC 100,APO_DIST 100,APO_FAC 50.0,ORI_TYP #VAR,CIRC_TYP #BASE,JERK_FAC 50.0}
DECL FDAT FP269={TOOL_NO 1,BASE_NO 2,IPO_FRAME #BASE,POINT2[] " ",TQ_STATE FALSE}
DECL E6POS XP269={X 501.05137,Y -625.26643,Z 815.36226,A -180,B 0,C 180,S 2,T 35,E1 0,E2 0,E3 0,E4 0,E5 0,E6 0}
DECL PDAT PPDATP92={VEL 100,ACC 100,APO_DIST 100,APO_MODE #CDIS,GEAR_JERK 100.000,EXAX_IGN 0}
DECL FDAT FP91={TOOL_NO 1,BASE_NO 2,IPO_FRAME #BASE,POINT2[] " ",TQ_STATE FALSE}
DECL E6POS XP91={X 463.27936,Y -81.1426,Z 1257.60001,A -90,B 0,C 180,S 2,T 35,E1 0,E2 0,E3 0,E4 0,E5 0,E6 0}
; DECL LDAT LCPDATP127={VEL 1,ACC 100,APO_DIST 100,APO_FAC 50.0,ORI_TYP #VAR,CIRC_TYP #BASE,JERK_FAC 50.0}
DECL FDAT FP681={TOOL_NO 1,BASE_NO 2,IPO_FRAME #BASE,POINT2[] " ",TQ_STATE FALSE}
DECL E6POS XP681={X 463.27964,Y -81.14297,Z 1127.60045,A -90,B 0,C 180,S 2,T 35,E1 0,E2 0,E3 0,E4 0,E5 0,E6 0}
; DECL LDAT LCPDATP126={VEL 1,ACC 100,APO_DIST 100,APO_FAC 50.0,ORI_TYP #VAR,CIRC_TYP #BASE,JERK_FAC 50.0}
DECL FDAT FP682={TOOL_NO 1,BASE_NO 2,IPO_FRAME #BASE,POINT2[] " ",TQ_STATE FALSE}
DECL E6POS XP682={X 463.28094,Y -31.14301,Z 1027.60139,A -90,B 0,C 180,S 2,T 35,E1 0,E2 0,E3 0,E4 0,E5 0,E6 0}
; DECL PDAT PPDATP64={VEL 100,ACC 100,APO_DIST 100,APO_MODE #CDIS,GEAR_JERK 100.000,EXAX_IGN 0}
DECL FDAT FP698={TOOL_NO 1,BASE_NO 2,IPO_FRAME #BASE,POINT2[] " ",TQ_STATE FALSE}
DECL E6POS XP698={X 463.28024,Y -561.1425,Z 1277.60113,A -90,B 0,C 180,S 2,T 35,E1 0,E2 0,E3 0,E4 0,E5 0,E6 0}
; DECL LDAT LCPDATP129={VEL 1,ACC 100,APO_DIST 100,APO_FAC 50.0,ORI_TYP #VAR,CIRC_TYP #BASE,JERK_FAC 50.0}
DECL FDAT FP699={TOOL_NO 1,BASE_NO 2,IPO_FRAME #BASE,POINT2[] " ",TQ_STATE FALSE}
DECL E6POS XP699={X 463.28024,Y -561.14273,Z 1177.60018,A -90,B 0,C 180,S 2,T 35,E1 0,E2 0,E3 0,E4 0,E5 0,E6 0}
; DECL LDAT LCPDATP128={VEL 1,ACC 100,APO_DIST 100,APO_FAC 50.0,ORI_TYP #VAR,CIRC_TYP #BASE,JERK_FAC 50.0}
DECL FDAT FP700={TOOL_NO 1,BASE_NO 2,IPO_FRAME #BASE,POINT2[] " ",TQ_STATE FALSE}
DECL E6POS XP700={X 463.28025,Y -511.14273,Z 1027.60074,A -90,B 0,C 180,S 2,T 35,E1 0,E2 0,E3 0,E4 0,E5 0,E6 0}
; DECL PDAT PPDATP65={VEL 100,ACC 100,APO_DIST 100,APO_MODE #CDIS,GEAR_JERK 100.000,EXAX_IGN 0}
DECL FDAT FP701={TOOL_NO 1,BASE_NO 2,IPO_FRAME #BASE,POINT2[] " ",TQ_STATE FALSE}
DECL E6POS XP701={X 866.03456,Y -625.26821,Z 1277.60068,A -180,B 0,C 180,S 2,T 35,E1 0,E2 0,E3 0,E4 0,E5 0,E6 0}
; DECL LDAT LCPDATP130={VEL 1,ACC 100,APO_DIST 100,APO_FAC 50.0,ORI_TYP #VAR,CIRC_TYP #BASE,JERK_FAC 50.0}
DECL FDAT FP702={TOOL_NO 1,BASE_NO 2,IPO_FRAME #BASE,POINT2[] " ",TQ_STATE FALSE}
DECL E6POS XP702={X 866.03456,Y -625.26838,Z 1177.59969,A 180,B 0,C 180,S 2,T 35,E1 0,E2 0,E3 0,E4 0,E5 0,E6 0}
; DECL LDAT LCPDATP131={VEL 1,ACC 100,APO_DIST 100,APO_FAC 50.0,ORI_TYP #VAR,CIRC_TYP #BASE,JERK_FAC 50.0}
DECL FDAT FP703={TOOL_NO 1,BASE_NO 2,IPO_FRAME #BASE,POINT2[] " ",TQ_STATE FALSE}
DECL E6POS XP703={X 816.03456,Y -625.26838,Z 1028.37539,A 180,B 0,C 180,S 2,T 35,E1 0,E2 0,E3 0,E4 0,E5 0,E6 0}
; DECL PDAT PPDATP66={VEL 100,ACC 100,APO_DIST 100,APO_MODE #CDIS,GEAR_JERK 100.000,EXAX_IGN 0}
DECL FDAT FP704={TOOL_NO 1,BASE_NO 2,IPO_FRAME #BASE,POINT2[] " ",TQ_STATE FALSE}
